C05383=1024.607,74.316,-103.652,167.758,48.129,158.923
C05384=1024.602,74.066,-103.634,167.757,48.134,158.924
C05385=1024.596,73.817,-103.616,167.754,48.137,158.924
C05386=1024.590,73.567,-103.600,167.751,48.141,158.924
C05387=1024.584,73.318,-103.582,167.749,48.146,158.925
C05388=1024.578,73.069,-103.565,167.746,48.150,158.925
C05389=1024.572,72.819,-103.547,167.743,48.154,158.926
C05390=1024.566,72.570,-103.530,167.740,48.157,158.926
C05391=1024.560,72.321,-103.512,167.739,48.162,158.926
C05392=1024.554,72.071,-103.494,167.736,48.166,158.927
C05393=1024.548,71.823,-103.477,167.733,48.169,158.927
C05394=1024.542,71.572,-103.460,167.730,48.173,158.928
C05395=1024.537,71.323,-103.443,167.728,48.178,158.928
C05396=1024.531,71.074,-103.425,167.725,48.182,158.928
C05397=1024.524,70.825,-103.408,167.723,48.185,158.929
C05398=1024.519,70.576,-103.390,167.721,48.190,158.929
C05399=1024.513,70.327,-103.372,167.718,48.194,158.930
C05400=1024.507,70.077,-103.356,167.715,48.197,158.930
C05401=1024.501,69.828,-103.338,167.712,48.201,158.930
C05402=1024.495,69.578,-103.320,167.710,48.206,158.931
C05403=1024.489,69.329,-103.303,167.708,48.209,158.931
C05404=1024.483,69.080,-103.286,167.705,48.213,158.932
C05405=1024.477,68.830,-103.269,167.702,48.217,158.932
C05406=1024.472,68.581,-103.251,167.700,48.222,158.933
C05407=1024.466,68.332,-103.234,167.697,48.226,158.933
C05408=1024.460,68.082,-103.217,167.694,48.229,158.933
C05409=1024.454,67.833,-103.200,167.692,48.234,158.934
C05410=1024.448,67.584,-103.182,167.690,48.238,158.934
C05411=1024.441,67.334,-103.165,167.687,48.241,158.935
C05412=1024.436,67.085,-103.148,167.684,48.245,158.935
C05413=1024.430,66.836,-103.131,167.682,48.250,158.935
C05414=1024.424,66.586,-103.113,167.679,48.254,158.936
C05415=1024.418,66.337,-103.097,167.676,48.258,158.936
C05416=1024.412,66.088,-103.079,167.674,48.262,158.937
C05417=1024.406,65.837,-103.062,167.672,48.266,158.937
C05418=1024.400,65.589,-103.045,167.669,48.270,158.937
C05419=1024.394,65.340,-103.028,167.667,48.274,158.938
C05420=1024.388,65.090,-103.011,167.664,48.278,158.938
C05421=1024.382,64.841,-102.993,167.661,48.282,158.939
C05422=1024.376,64.592,-102.976,167.658,48.286,158.939
C05423=1024.370,64.342,-102.959,167.656,48.290,158.940
C05424=1024.364,64.093,-102.942,167.654,48.294,158.940
C05425=1024.359,63.843,-102.925,167.651,48.298,158.940
C05426=1024.352,63.594,-102.908,167.649,48.302,158.941
C05427=1024.347,63.344,-102.891,167.646,48.306,158.941
C05428=1024.341,63.095,-102.874,167.643,48.310,158.942
C05429=1024.334,62.845,-102.858,167.641,48.315,158.942
C05430=1024.328,62.597,-102.841,167.638,48.319,158.942
C05431=1024.323,62.347,-102.824,167.635,48.323,158.943
C05432=1024.317,62.098,-102.808,167.633,48.327,158.943
C05433=1024.310,61.848,-102.790,167.631,48.331,158.944
C05434=1024.304,61.599,-102.774,167.628,48.335,158.944
C05435=1024.298,61.350,-102.757,167.626,48.339,158.945
C05436=1024.292,61.100,-102.740,167.623,48.344,158.945
C05437=1024.285,60.851,-102.723,167.620,48.347,158.945
C05438=1024.279,60.602,-102.707,167.618,48.352,158.946
C05439=1024.274,60.352,-102.690,167.615,48.356,158.946
C05440=1024.267,60.103,-102.673,167.612,48.360,158.947
C05441=1024.260,59.819,-102.654,167.610,48.364,158.947
C05442=1024.253,59.534,-102.635,167.606,48.369,158.948
C05443=1024.246,59.249,-102.616,167.604,48.374,158.948
C05444=1024.240,58.965,-102.596,167.600,48.379,158.948
C05445=1024.234,58.716,-102.580,167.598,48.383,158.949
C05446=1024.227,58.466,-102.564,167.595,48.387,158.949
C05447=1024.221,58.217,-102.547,167.594,48.391,158.950
C05448=1024.215,57.967,-102.530,167.591,48.395,158.950
C05449=1024.209,57.718,-102.514,167.588,48.399,158.951
C05450=1024.204,57.469,-102.497,167.585,48.404,158.951
C05451=1024.197,57.219,-102.480,167.583,48.408,158.952
C05452=1024.191,56.970,-102.464,167.580,48.412,158.952
C05453=1024.185,56.721,-102.447,167.577,48.416,158.952
C05454=1024.179,56.472,-102.430,167.575,48.420,158.953
C05455=1024.174,56.222,-102.414,167.572,48.424,158.953
C05456=1024.167,55.972,-102.397,167.569,48.428,158.954
C05457=1024.161,55.723,-102.380,167.568,48.432,158.954
C05458=1024.155,55.474,-102.364,167.565,48.436,158.954
C05459=1024.149,55.224,-102.347,167.562,48.441,158.955
C05460=1024.143,54.975,-102.331,167.560,48.444,158.955
C05461=1024.137,54.725,-102.313,167.557,48.448,158.956
C05462=1024.131,54.476,-102.297,167.554,48.453,158.956
C05463=1024.125,54.227,-102.281,167.551,48.457,158.956
C05464=1024.119,53.977,-102.264,167.549,48.461,158.957
C05465=1024.113,53.728,-102.248,167.547,48.465,158.957
C05466=1024.107,53.479,-102.231,167.544,48.469,158.958
C05467=1024.102,53.230,-102.214,167.542,48.473,158.958
C05468=1024.095,52.980,-102.198,167.539,48.477,158.958
C05469=1024.089,52.730,-102.182,167.536,48.481,158.959
C05470=1024.083,52.481,-102.165,167.534,48.485,158.959
C05471=1024.077,52.232,-102.148,167.531,48.489,158.960
C05472=1024.071,51.983,-102.132,167.528,48.494,158.960
C05473=1024.066,51.733,-102.115,167.527,48.497,158.961
C05474=1024.060,51.484,-102.099,167.524,48.501,158.961
C05475=1024.054,51.234,-102.083,167.521,48.505,158.961
C05476=1024.048,50.985,-102.066,167.519,48.510,158.962
C05477=1024.041,50.735,-102.050,167.516,48.513,158.962
C05478=1024.035,50.486,-102.033,167.513,48.517,158.962
C05479=1024.030,50.237,-102.016,167.510,48.521,158.963
C05480=1024.024,49.987,-102.000,167.508,48.525,158.963
C05481=1024.018,49.738,-101.983,167.506,48.529,158.964
C05482=1024.012,49.489,-101.967,167.503,48.533,158.964
C05483=1024.006,49.239,-101.951,167.500,48.537,158.964
C05484=1024.000,48.990,-101.935,167.498,48.541,158.965
C05485=1023.995,48.740,-101.918,167.495,48.546,158.965
C05486=1023.989,48.491,-101.902,167.493,48.549,158.966
C05487=1023.983,48.242,-101.885,167.491,48.553,158.966
C05488=1023.977,47.992,-101.869,167.488,48.557,158.966
C05489=1023.971,47.743,-101.853,167.485,48.561,158.967
C05490=1023.965,47.494,-101.836,167.483,48.566,158.967
C05491=1023.959,47.245,-101.820,167.480,48.570,158.968
C05492=1023.954,46.995,-101.803,167.478,48.573,158.968
C05493=1023.948,46.746,-101.786,167.475,48.577,158.968
C05494=1023.942,46.496,-101.770,167.472,48.581,158.969
C05495=1023.935,46.246,-101.754,167.470,48.585,158.969
C05496=1023.929,45.997,-101.737,167.467,48.589,158.969
C05497=1023.923,45.748,-101.721,167.464,48.593,158.970
C05498=1023.917,45.498,-101.705,167.463,48.597,158.970
C05499=1023.912,45.249,-101.688,167.460,48.601,158.971
C05500=1023.906,44.999,-101.672,167.457,48.605,158.971
C05501=1023.901,44.751,-101.656,167.454,48.609,158.971
C05502=1023.895,44.501,-101.640,167.452,48.613,158.972
C05503=1023.889,44.252,-101.623,167.449,48.617,158.972
C05504=1023.883,44.003,-101.607,167.447,48.621,158.973
C05505=1023.876,43.717,-101.589,167.444,48.625,158.973
C05506=1023.870,43.433,-101.570,167.441,48.630,158.973
C05507=1023.863,43.148,-101.551,167.439,48.634,158.974
C05508=1023.857,42.863,-101.533,167.435,48.638,158.974
C05509=1023.851,42.614,-101.516,167.432,48.642,158.974
C05510=1023.845,42.364,-101.501,167.431,48.647,158.975
C05511=1023.839,42.115,-101.484,167.428,48.651,158.975
C05512=1023.833,41.865,-101.469,167.425,48.654,158.976
C05513=1023.827,41.616,-101.453,167.422,48.658,158.976
C05514=1023.821,41.366,-101.436,167.420,48.663,158.977
C05515=1023.815,41.117,-101.420,167.417,48.667,158.977
C05516=1023.809,40.868,-101.404,167.414,48.671,158.977
C05517=1023.804,40.618,-101.388,167.412,48.675,158.978
C05518=1023.797,40.369,-101.373,167.409,48.679,158.978
C05519=1023.791,40.119,-101.356,167.407,48.683,158.978
C05520=1023.785,39.870,-101.340,167.405,48.687,158.979
C05521=1023.779,39.620,-101.325,167.402,48.691,158.979
C05522=1023.773,39.371,-101.308,167.399,48.695,158.980
C05523=1023.767,39.121,-101.292,167.397,48.699,158.980
C05524=1023.761,38.872,-101.276,167.394,48.703,158.980
C05525=1023.756,38.623,-101.261,167.391,48.707,158.981
C05526=1023.750,38.374,-101.245,167.388,48.711,158.981
C05527=1023.744,38.124,-101.229,167.387,48.715,158.982
C05528=1023.738,37.874,-101.213,167.384,48.719,158.982
C05529=1023.732,37.625,-101.197,167.381,48.723,158.982
C05530=1023.726,37.376,-101.181,167.378,48.727,158.983
C05531=1023.720,37.126,-101.166,167.376,48.731,158.983
C05532=1023.714,36.877,-101.150,167.373,48.736,158.983
C05533=1023.708,36.627,-101.133,167.370,48.740,158.984
C05534=1023.702,36.377,-101.118,167.368,48.744,158.984
C05535=1023.696,36.129,-101.102,167.365,48.747,158.984
C05536=1023.691,35.879,-101.087,167.363,48.752,158.985
C05537=1023.684,35.630,-101.071,167.361,48.756,158.985
C05538=1023.678,35.380,-101.056,167.358,48.760,158.986
C05539=1023.672,35.131,-101.039,167.356,48.764,158.986
C05540=1023.666,34.881,-101.025,167.353,48.768,158.987
C05541=1023.660,34.632,-101.008,167.350,48.772,158.987
C05542=1023.654,34.382,-100.993,167.348,48.777,158.987
C05543=1023.648,34.133,-100.977,167.345,48.781,158.988
C05544=1023.643,33.883,-100.962,167.342,48.785,158.988
C05545=1023.636,33.634,-100.946,167.339,48.789,158.988
C05546=1023.630,33.384,-100.931,167.337,48.793,158.989
C05547=1023.624,33.135,-100.915,167.334,48.797,158.989
C05548=1023.618,32.885,-100.899,167.331,48.801,158.990
C05549=1023.612,32.636,-100.883,167.329,48.805,158.990
C05550=1023.606,32.387,-100.869,167.327,48.809,158.991
C05551=1023.600,32.138,-100.852,167.324,48.813,158.991
C05552=1023.594,31.888,-100.837,167.322,48.817,158.991
C05553=1023.588,31.639,-100.821,167.319,48.821,158.992
C05554=1023.582,31.389,-100.806,167.316,48.826,158.992
C05555=1023.576,31.141,-100.790,167.314,48.830,158.992
C05556=1023.571,30.891,-100.775,167.311,48.834,158.993
C05557=1023.564,30.641,-100.760,167.308,48.837,158.993
C05558=1023.558,30.392,-100.744,167.305,48.841,158.993
C05559=1023.553,30.142,-100.728,167.303,48.846,158.994
C05560=1023.546,29.893,-100.713,167.300,48.850,158.994
C05561=1023.541,29.643,-100.697,167.298,48.854,158.995
C05562=1023.534,29.394,-100.682,167.296,48.858,158.995
C05563=1023.528,29.144,-100.666,167.293,48.861,158.995
C05564=1023.523,28.894,-100.650,167.290,48.866,158.996
C05565=1023.517,28.645,-100.636,167.288,48.870,158.996
C05566=1023.511,28.396,-100.620,167.285,48.874,158.996
C05567=1023.505,28.146,-100.605,167.282,48.878,158.997
C05568=1023.499,27.897,-100.588,167.279,48.882,158.997
C05569=1023.492,27.612,-100.572,167.277,48.887,158.998
C05570=1023.485,27.327,-100.555,167.273,48.891,158.998
C05571=1023.479,27.043,-100.537,167.271,48.896,158.999
C05572=1023.472,26.758,-100.519,167.268,48.901,158.999
C05573=1023.466,26.508,-100.504,167.265,48.905,158.999
C05574=1023.460,26.259,-100.488,167.262,48.909,159.000
C05575=1023.453,26.009,-100.473,167.259,48.913,159.000
C05576=1023.448,25.760,-100.458,167.257,48.917,159.000
C05577=1023.442,25.510,-100.443,167.255,48.921,159.001
C05578=1023.435,25.261,-100.427,167.252,48.925,159.001
C05579=1023.430,25.011,-100.412,167.250,48.929,159.002
C05580=1023.424,24.762,-100.397,167.247,48.934,159.002
C05581=1023.417,24.513,-100.382,167.244,48.938,159.002
C05582=1023.412,24.263,-100.367,167.242,48.942,159.003
C05583=1023.406,24.014,-100.352,167.239,48.945,159.003
C05584=1023.399,23.765,-100.337,167.237,48.950,159.004
C05585=1023.394,23.515,-100.321,167.234,48.954,159.004
C05586=1023.388,23.266,-100.306,167.231,48.958,159.004
C05587=1023.381,23.016,-100.291,167.228,48.962,159.005
C05588=1023.376,22.766,-100.276,167.226,48.967,159.005
C05589=1023.369,22.517,-100.261,167.223,48.971,159.005
C05590=1023.364,22.268,-100.246,167.220,48.974,159.006
C05591=1023.358,22.018,-100.231,167.218,48.978,159.006
C05592=1023.352,21.768,-100.216,167.215,48.982,159.006
C05593=1023.346,21.520,-100.201,167.212,48.987,159.007
C05594=1023.340,21.270,-100.185,167.210,48.991,159.007
C05595=1023.334,21.020,-100.170,167.207,48.995,159.008
C05596=1023.328,20.771,-100.156,167.205,48.999,159.008
C05597=1023.322,20.521,-100.140,167.202,49.003,159.008
C05598=1023.316,20.272,-100.125,167.200,49.006,159.009
C05599=1023.310,20.023,-100.110,167.197,49.011,159.009
C05600=1023.304,19.773,-100.095,167.194,49.015,159.009
C05601=1023.299,19.524,-100.080,167.192,49.019,159.010
C05602=1023.292,19.274,-100.065,167.189,49.023,159.010
C05603=1023.286,19.024,-100.050,167.186,49.027,159.010
C05604=1023.281,18.775,-100.035,167.184,49.032,159.011
C05605=1023.274,18.525,-100.020,167.181,49.036,159.011
C05606=1023.268,18.276,-100.005,167.178,49.039,159.012
C05607=1023.262,18.027,-99.991,167.175,49.043,159.012
C05608=1023.257,17.777,-99.975,167.173,49.047,159.012
C05609=1023.251,17.528,-99.961,167.170,49.052,159.013
C05610=1023.245,17.278,-99.946,167.168,49.056,159.013
C05611=1023.238,17.028,-99.932,167.165,49.060,159.013
C05612=1023.232,16.779,-99.917,167.162,49.064,159.014
C05613=1023.226,16.529,-99.902,167.160,49.069,159.014
C05614=1023.221,16.280,-99.887,167.157,49.073,159.015
C05615=1023.215,16.030,-99.872,167.154,49.077,159.015
C05616=1023.209,15.781,-99.857,167.151,49.080,159.015
C05617=1023.203,15.532,-99.842,167.149,49.084,159.015
C05618=1023.196,15.282,-99.827,167.146,49.088,159.016
C05619=1023.191,15.032,-99.813,167.144,49.093,159.016
C05620=1023.185,14.783,-99.798,167.142,49.097,159.017
C05621=1023.179,14.534,-99.783,167.139,49.101,159.017
C05622=1023.173,14.284,-99.768,167.136,49.105,159.017
C05623=1023.167,14.035,-99.754,167.134,49.109,159.018
C05624=1023.161,13.785,-99.739,167.131,49.113,159.018
C05625=1023.156,13.535,-99.724,167.128,49.117,159.018
C05626=1023.150,13.286,-99.710,167.126,49.121,159.019
C05627=1023.142,13.036,-99.695,167.123,49.125,159.019
C05628=1023.137,12.787,-99.681,167.120,49.129,159.020
C05629=1023.131,12.537,-99.666,167.118,49.134,159.020
C05630=1023.125,12.288,-99.652,167.115,49.138,159.020
C05631=1023.119,12.038,-99.638,167.112,49.142,159.021
C05632=1023.113,11.789,-99.623,167.109,49.147,159.021
C05633=1023.106,11.506,-99.607,167.106,49.151,159.021
C05634=1023.099,11.222,-99.590,167.103,49.156,159.022
C05635=1023.092,10.939,-99.574,167.100,49.160,159.022
C05636=1023.085,10.656,-99.558,167.097,49.165,159.023
C05637=1023.079,10.406,-99.543,167.094,49.169,159.023
C05638=1023.073,10.157,-99.528,167.092,49.174,159.024
C05639=1023.067,9.907,-99.514,167.089,49.178,159.024
C05640=1023.061,9.658,-99.500,167.086,49.182,159.024
C05641=1023.055,9.408,-99.485,167.083,49.186,159.024
C05642=1023.049,9.159,-99.471,167.081,49.190,159.025
C05643=1023.043,8.909,-99.456,167.078,49.194,159.025
C05644=1023.037,8.660,-99.442,167.076,49.198,159.026
C05645=1023.030,8.410,-99.428,167.073,49.202,159.026
C05646=1023.025,8.161,-99.414,167.070,49.207,159.026
C05647=1023.018,7.911,-99.399,167.068,49.211,159.027
C05648=1023.013,7.662,-99.384,167.065,49.215,159.027
C05649=1023.007,7.412,-99.370,167.062,49.219,159.027
C05650=1023.001,7.163,-99.355,167.059,49.223,159.028
C05651=1022.995,6.913,-99.341,167.057,49.228,159.028
C05652=1022.989,6.664,-99.327,167.054,49.232,159.029
C05653=1022.984,6.414,-99.313,167.052,49.236,159.029
C05654=1022.976,6.165,-99.298,167.049,49.240,159.029
C05655=1022.971,5.915,-99.285,167.046,49.244,159.030
C05656=1022.965,5.665,-99.270,167.044,49.248,159.030
C05657=1022.959,5.416,-99.256,167.041,49.252,159.030
C05658=1022.953,5.167,-99.241,167.038,49.256,159.031
C05659=1022.947,4.917,-99.227,167.035,49.260,159.031
C05660=1022.941,4.668,-99.212,167.033,49.264,159.031
C05661=1022.935,4.417,-99.198,167.030,49.268,159.032
C05662=1022.929,4.169,-99.184,167.027,49.272,159.032
C05663=1022.923,3.919,-99.170,167.025,49.277,159.032
C05664=1022.917,3.669,-99.156,167.022,49.281,159.033
C05665=1022.911,3.420,-99.141,167.019,49.285,159.033
C05666=1022.905,3.170,-99.127,167.017,49.289,159.033
C05667=1022.900,2.921,-99.113,167.014,49.293,159.034
C05668=1022.894,2.671,-99.099,167.011,49.297,159.034
C05669=1022.887,2.421,-99.085,167.008,49.301,159.034
C05670=1022.882,2.172,-99.071,167.006,49.305,159.035
C05671=1022.876,1.923,-99.057,167.003,49.309,159.035
C05672=1022.870,1.673,-99.042,167.001,49.313,159.035
C05673=1022.864,1.423,-99.028,166.998,49.317,159.036
C05674=1022.859,1.174,-99.014,166.995,49.321,159.036
C05675=1022.852,0.924,-98.999,166.992,49.325,159.036
C05676=1022.846,0.675,-98.986,166.990,49.329,159.037
C05677=1022.841,0.425,-98.972,166.987,49.333,159.037
C05678=1022.834,0.176,-98.957,166.984,49.337,159.037
C05679=1022.829,-0.074,-98.943,166.981,49.341,159.038
C05680=1022.823,-0.324,-98.929,166.979,49.345,159.038
C05681=1022.818,-0.572,-98.915,166.976,49.349,159.038
C05682=1022.811,-0.823,-98.900,166.973,49.353,159.039
C05683=1022.805,-1.072,-98.887,166.970,49.357,159.039
C05684=1022.799,-1.321,-98.873,166.968,49.361,159.039
C05685=1022.793,-1.571,-98.858,166.965,49.365,159.040
C05686=1022.788,-1.821,-98.845,166.962,49.369,159.040
C05687=1022.782,-2.070,-98.830,166.960,49.373,159.040
C05688=1022.777,-2.319,-98.816,166.957,49.377,159.041
C05689=1022.771,-2.570,-98.802,166.954,49.381,159.041
C05690=1022.764,-2.819,-98.789,166.951,49.385,159.041
C05691=1022.759,-3.068,-98.774,166.949,49.389,159.042
C05692=1022.753,-3.317,-98.760,166.946,49.393,159.042
C05693=1022.747,-3.568,-98.746,166.943,49.397,159.042
C05694=1022.742,-3.817,-98.732,166.940,49.401,159.042
C05695=1022.736,-4.067,-98.718,166.938,49.405,159.043
C05696=1022.730,-4.315,-98.704,166.935,49.410,159.043
C05697=1022.722,-4.598,-98.689,166.932,49.414,159.043
C05698=1022.715,-4.879,-98.673,166.928,49.419,159.044
C05699=1022.709,-5.161,-98.658,166.926,49.424,159.044
C05700=1022.702,-5.442,-98.642,166.922,49.429,159.045
C05701=1022.696,-5.691,-98.628,166.920,49.433,159.045
C05702=1022.690,-5.941,-98.615,166.917,49.437,159.045
C05703=1022.685,-6.190,-98.601,166.914,49.441,159.046
C05704=1022.678,-6.440,-98.588,166.911,49.445,159.046
C05705=1022.672,-6.690,-98.574,166.909,49.449,159.047
C05706=1022.666,-6.939,-98.561,166.906,49.453,159.047
C05707=1022.661,-7.189,-98.547,166.904,49.457,159.047
C05708=1022.655,-7.438,-98.533,166.900,49.462,159.047
C05709=1022.648,-7.688,-98.519,166.897,49.466,159.048
C05710=1022.642,-7.937,-98.506,166.894,49.470,159.048
C05711=1022.637,-8.187,-98.492,166.892,49.474,159.048
C05712=1022.631,-8.436,-98.479,166.889,49.478,159.049
C05713=1022.625,-8.686,-98.465,166.887,49.482,159.049
C05714=1022.619,-8.935,-98.452,166.884,49.486,159.049
C05715=1022.613,-9.185,-98.437,166.881,49.490,159.050
C05716=1022.607,-9.435,-98.424,166.878,49.495,159.050
C05717=1022.601,-9.685,-98.411,166.876,49.499,159.050
C05718=1022.595,-9.934,-98.398,166.873,49.503,159.051
C05719=1022.590,-10.184,-98.384,166.871,49.507,159.051
C05720=1022.583,-10.433,-98.371,166.867,49.512,159.051
C05721=1022.577,-10.682,-98.357,166.864,49.516,159.052
C05722=1022.571,-10.933,-98.343,166.861,49.520,159.052
C05723=1022.565,-11.182,-98.330,166.859,49.524,159.052
C05724=1022.559,-11.431,-98.316,166.856,49.528,159.053
C05725=1022.553,-11.681,-98.303,166.853,49.532,159.053
C05726=1022.548,-11.930,-98.289,166.851,49.536,159.053
C05727=1022.542,-12.180,-98.276,166.848,49.540,159.054
C05728=1022.536,-12.430,-98.262,166.845,49.544,159.054
C05729=1022.530,-12.679,-98.249,166.842,49.548,159.054
C05730=1022.525,-12.928,-98.235,166.840,49.552,159.054
C05731=1022.518,-13.178,-98.222,166.837,49.556,159.055
C05732=1022.512,-13.428,-98.208,166.835,49.560,159.055
C05733=1022.507,-13.678,-98.195,166.832,49.564,159.056
C05734=1022.501,-13.928,-98.181,166.828,49.569,159.056
C05735=1022.495,-14.177,-98.168,166.825,49.573,159.056
C05736=1022.489,-14.426,-98.155,166.823,49.577,159.056
C05737=1022.483,-14.676,-98.141,166.820,49.581,159.057
C05738=1022.477,-14.925,-98.128,166.817,49.585,159.057
C05739=1022.472,-15.175,-98.115,166.814,49.589,159.057
C05740=1022.466,-15.424,-98.101,166.812,49.593,159.058
C05741=1022.460,-15.674,-98.087,166.809,49.597,159.058
C05742=1022.454,-15.924,-98.075,166.806,49.601,159.058
C05743=1022.448,-16.173,-98.062,166.804,49.605,159.059
C05744=1022.442,-16.422,-98.048,166.801,49.609,159.059
C05745=1022.437,-16.673,-98.035,166.797,49.613,159.059
C05746=1022.430,-16.922,-98.022,166.795,49.618,159.060
C05747=1022.424,-17.172,-98.009,166.792,49.622,159.060
C05748=1022.418,-17.421,-97.996,166.789,49.626,159.060
C05749=1022.412,-17.670,-97.983,166.787,49.630,159.061
C05750=1022.407,-17.920,-97.970,166.784,49.634,159.061
C05751=1022.401,-18.170,-97.956,166.781,49.638,159.061
C05752=1022.395,-18.420,-97.944,166.777,49.642,159.061
C05753=1022.389,-18.669,-97.931,166.775,49.647,159.062
C05754=1022.383,-18.919,-97.918,166.772,49.651,159.062
C05755=1022.377,-19.168,-97.904,166.770,49.655,159.062
C05756=1022.371,-19.417,-97.891,166.767,49.659,159.063
C05757=1022.365,-19.667,-97.878,166.764,49.663,159.063
C05758=1022.359,-19.917,-97.865,166.762,49.667,159.063
C05759=1022.353,-20.167,-97.852,166.758,49.671,159.064
C05760=1022.347,-20.416,-97.839,166.755,49.675,159.064
C05761=1022.340,-20.696,-97.824,166.753,49.680,159.064
C05762=1022.334,-20.976,-97.809,166.749,49.685,159.065
C05763=1022.327,-21.255,-97.795,166.746,49.690,159.065
C05764=1022.320,-21.535,-97.780,166.743,49.694,159.065
C05765=1022.314,-21.785,-97.768,166.740,49.698,159.066
C05766=1022.309,-22.035,-97.755,166.738,49.702,159.066
C05767=1022.302,-22.284,-97.742,166.734,49.707,159.066
C05768=1022.297,-22.533,-97.730,166.731,49.711,159.067
C05769=1022.292,-22.783,-97.716,166.729,49.715,159.067
C05770=1022.286,-23.033,-97.703,166.726,49.719,159.067
C05771=1022.279,-23.282,-97.690,166.723,49.723,159.067
C05772=1022.274,-23.532,-97.677,166.720,49.727,159.068
C05773=1022.267,-23.781,-97.664,166.718,49.731,159.068
C05774=1022.261,-24.031,-97.652,166.715,49.735,159.068
C05775=1022.256,-24.281,-97.638,166.711,49.739,159.069
C05776=1022.250,-24.530,-97.625,166.709,49.743,159.069
C05777=1022.244,-24.780,-97.613,166.706,49.747,159.069
C05778=1022.238,-25.029,-97.600,166.703,49.751,159.069
C05779=1022.233,-25.279,-97.587,166.700,49.755,159.070
C05780=1022.227,-25.529,-97.575,166.698,49.759,159.070
C05781=1022.221,-25.778,-97.561,166.695,49.763,159.070
C05782=1022.215,-26.028,-97.548,166.692,49.767,159.071
C05783=1022.209,-26.278,-97.536,166.689,49.772,159.071
C05784=1022.204,-26.527,-97.523,166.686,49.776,159.071
C05785=1022.198,-26.776,-97.510,166.683,49.780,159.072
C05786=1022.192,-27.026,-97.498,166.681,49.784,159.072
C05787=1022.186,-27.276,-97.484,166.678,49.788,159.072
C05788=1022.181,-27.526,-97.471,166.675,49.792,159.072
C05789=1022.175,-27.776,-97.459,166.672,49.796,159.073
C05790=1022.168,-28.025,-97.447,166.669,49.800,159.073
C05791=1022.163,-28.274,-97.435,166.666,49.804,159.073
C05792=1022.156,-28.524,-97.421,166.664,49.809,159.074
C05793=1022.151,-28.774,-97.409,166.661,49.813,159.074
C05794=1022.145,-29.023,-97.396,166.658,49.817,159.074
C05795=1022.139,-29.273,-97.384,166.654,49.822,159.074
C05796=1022.133,-29.523,-97.371,166.652,49.826,159.075
C05797=1022.128,-29.772,-97.359,166.649,49.830,159.075
C05798=1022.122,-30.022,-97.346,166.646,49.834,159.075
C05799=1022.115,-30.271,-97.334,166.644,49.838,159.076
C05800=1022.109,-30.521,-97.321,166.641,49.842,159.076
C05801=1022.103,-30.770,-97.309,166.638,49.847,159.076
C05802=1022.098,-31.020,-97.296,166.635,49.851,159.077
C05803=1022.092,-31.270,-97.284,166.632,49.855,159.077
C05804=1022.086,-31.520,-97.271,166.629,49.859,159.077
C05805=1022.080,-31.770,-97.259,166.627,49.863,159.078
C05806=1022.075,-32.019,-97.246,166.623,49.867,159.078
C05807=1022.068,-32.269,-97.235,166.620,49.871,159.078
C05808=1022.062,-32.518,-97.222,166.618,49.875,159.078
C05809=1022.057,-32.768,-97.210,166.615,49.880,159.079
C05810=1022.051,-33.018,-97.197,166.612,49.884,159.079
C05811=1022.045,-33.267,-97.184,166.608,49.888,159.079
C05812=1022.039,-33.517,-97.171,166.606,49.892,159.079
C05813=1022.033,-33.766,-97.159,166.603,49.896,159.080
C05814=1022.027,-34.015,-97.147,166.600,49.900,159.080
C05815=1022.021,-34.265,-97.135,166.598,49.904,159.080
C05816=1022.015,-34.514,-97.123,166.594,49.908,159.081
C05817=1022.010,-34.764,-97.110,166.591,49.913,159.081
C05818=1022.004,-35.014,-97.097,166.589,49.917,159.081
C05819=1021.998,-35.263,-97.085,166.586,49.921,159.081
C05820=1021.992,-35.513,-97.073,166.583,49.925,159.082
C05821=1021.986,-35.764,-97.061,166.580,49.929,159.082
C05822=1021.981,-36.013,-97.049,166.577,49.933,159.082
C05823=1021.975,-36.263,-97.037,166.574,49.937,159.083
C05824=1021.969,-36.512,-97.024,166.571,49.941,159.083
C05825=1021.962,-36.791,-97.011,166.568,49.946,159.083
C05826=1021.956,-37.070,-96.996,166.565,49.950,159.084
C05827=1021.949,-37.349,-96.983,166.562,49.955,159.084
C05828=1021.943,-37.627,-96.969,166.558,49.960,159.084
C05829=1021.938,-37.878,-96.957,166.555,49.964,159.084
C05830=1021.932,-38.127,-96.945,166.553,49.968,159.085
C05831=1021.926,-38.376,-96.933,166.550,49.972,159.085
C05832=1021.920,-38.626,-96.920,166.547,49.976,159.085
C05833=1021.915,-38.876,-96.908,166.545,49.980,159.086
C05834=1021.909,-39.125,-96.895,166.541,49.984,159.086
C05835=1021.903,-39.375,-96.883,166.538,49.988,159.086
C05836=1021.897,-39.625,-96.872,166.536,49.993,159.086
C05837=1021.891,-39.875,-96.859,166.533,49.997,159.087
C05838=1021.885,-40.124,-96.848,166.529,50.001,159.087
C05839=1021.880,-40.374,-96.836,166.526,50.005,159.087
C05840=1021.873,-40.624,-96.824,166.524,50.009,159.087
C05841=1021.868,-40.873,-96.812,166.521,50.013,159.088
C05842=1021.862,-41.123,-96.799,166.517,50.018,159.088
C05843=1021.856,-41.372,-96.788,166.515,50.022,159.088
C05844=1021.850,-41.622,-96.776,166.512,50.026,159.089
C05845=1021.844,-41.871,-96.764,166.510,50.030,159.089
C05846=1021.838,-42.121,-96.753,166.506,50.035,159.089
C05847=1021.832,-42.371,-96.740,166.503,50.039,159.089
C05848=1021.826,-42.620,-96.728,166.501,50.043,159.090
C05849=1021.821,-42.871,-96.717,166.498,50.047,159.090
C05850=1021.815,-43.120,-96.705,166.494,50.051,159.090
C05851=1021.809,-43.369,-96.692,166.491,50.055,159.091
C05852=1021.803,-43.619,-96.681,166.489,50.059,159.091
C05853=1021.797,-43.869,-96.669,166.486,50.064,159.091
C05854=1021.792,-44.119,-96.657,166.483,50.068,159.091
C05855=1021.786,-44.368,-96.646,166.480,50.072,159.092
C05856=1021.780,-44.617,-96.633,166.477,50.076,159.092
C05857=1021.774,-44.868,-96.622,166.474,50.080,159.092
C05858=1021.769,-45.117,-96.610,166.472,50.084,159.092
C05859=1021.762,-45.367,-96.599,166.468,50.089,159.093
C05860=1021.757,-45.616,-96.586,166.465,50.093,159.093
C05861=1021.751,-45.866,-96.575,166.462,50.097,159.093
C05862=1021.745,-46.115,-96.563,166.460,50.101,159.094
C05863=1021.740,-46.366,-96.551,166.456,50.105,159.094
C05864=1021.734,-46.615,-96.540,166.453,50.109,159.094
C05865=1021.728,-46.865,-96.527,166.451,50.113,159.094
C05866=1021.722,-47.114,-96.516,166.448,50.117,159.095
C05867=1021.717,-47.363,-96.504,166.445,50.121,159.095
C05868=1021.710,-47.614,-96.493,166.442,50.126,159.095
C05869=1021.705,-47.863,-96.481,166.439,50.130,159.095
C05870=1021.699,-48.113,-96.469,166.436,50.134,159.096
C05871=1021.693,-48.362,-96.457,166.434,50.138,159.096
C05872=1021.688,-48.613,-96.445,166.430,50.142,159.096
C05873=1021.682,-48.862,-96.434,166.427,50.147,159.096
C05874=1021.677,-49.111,-96.422,166.424,50.150,159.097
C05875=1021.670,-49.362,-96.411,166.421,50.154,159.097
C05876=1021.665,-49.611,-96.399,166.419,50.158,159.097
C05877=1021.659,-49.861,-96.388,166.415,50.162,159.097
C05878=1021.653,-50.110,-96.375,166.412,50.167,159.098
C05879=1021.648,-50.360,-96.364,166.410,50.171,159.098
C05880=1021.642,-50.610,-96.353,166.407,50.175,159.098
C05881=1021.636,-50.859,-96.341,166.403,50.179,159.098
C05882=1021.631,-51.109,-96.330,166.401,50.183,159.099
C05883=1021.625,-51.359,-96.318,166.398,50.187,159.099
C05884=1021.619,-51.608,-96.307,166.394,50.192,159.099
C05885=1021.612,-51.858,-96.295,166.392,50.196,159.099
C05886=1021.607,-52.107,-96.285,166.389,50.201,159.100
C05887=1021.602,-52.357,-96.273,166.385,50.205,159.100
C05888=1021.595,-52.607,-96.262,166.383,50.209,159.100
C05889=1021.589,-52.855,-96.251,166.380,50.213,159.101
C05890=1021.583,-53.103,-96.239,166.376,50.217,159.101
C05891=1021.578,-53.350,-96.229,166.374,50.222,159.101
C05892=1021.572,-53.597,-96.217,166.371,50.226,159.101
C05893=1021.566,-53.845,-96.206,166.368,50.231,159.102
C05894=1021.560,-54.093,-96.195,166.365,50.235,159.102
C05895=1021.554,-54.341,-96.185,166.362,50.239,159.102
C05896=1021.548,-54.589,-96.173,166.360,50.243,159.103
C05897=1021.543,-54.838,-96.162,166.356,50.247,159.103
C05898=1021.537,-55.088,-96.151,166.353,50.251,159.103
C05899=1021.531,-55.338,-96.140,166.351,50.256,159.103
C05900=1021.525,-55.587,-96.129,166.347,50.260,159.103
C05901=1021.520,-55.837,-96.117,166.344,50.264,159.104
C05902=1021.514,-56.087,-96.106,166.342,50.268,159.104
C05903=1021.508,-56.337,-96.095,166.338,50.273,159.104
C05904=1021.502,-56.586,-96.084,166.335,50.277,159.105
C05905=1021.496,-56.835,-96.073,166.333,50.281,159.105
C05906=1021.490,-57.085,-96.062,166.329,50.286,159.105
C05907=1021.484,-57.335,-96.051,166.326,50.290,159.105
C05908=1021.478,-57.584,-96.040,166.324,50.294,159.106
C05909=1021.472,-57.868,-96.027,166.320,50.299,159.106
C05910=1021.465,-58.151,-96.015,166.317,50.304,159.106
C05911=1021.459,-58.434,-96.002,166.313,50.309,159.107
C05912=1021.452,-58.717,-95.990,166.310,50.313,159.107
C05913=1021.447,-58.968,-95.978,166.307,50.317,159.107
C05914=1021.441,-59.217,-95.967,166.303,50.322,159.107
///RCONF 1,0,0,1,0,0,0,0,0,0,0,0,0,0,0,0,0,0,0,0,0,0,0,0
C05915=1021.435,-59.467,-95.956,166.301,50.326,159.108
C05916=1021.429,-59.716,-95.945,166.298,50.330,159.108
C05917=1021.424,-59.966,-95.935,166.294,50.334,159.108
C05918=1021.417,-60.216,-95.923,166.292,50.338,159.108
C05919=1021.411,-60.465,-95.912,166.289,50.342,159.109
C05920=1021.406,-60.715,-95.902,166.285,50.347,159.109
C05921=1021.401,-60.964,-95.890,166.283,50.352,159.109
C05922=1021.395,-61.214,-95.879,166.280,50.356,159.110
C05923=1021.389,-61.463,-95.868,166.277,50.359,159.110
C05924=1021.383,-61.714,-95.858,166.273,50.363,159.110
C05925=1021.377,-61.964,-95.847,166.271,50.368,159.110
C05926=1021.372,-62.213,-95.836,166.268,50.372,159.110
C05927=1021.366,-62.463,-95.825,166.264,50.376,159.111
C05928=1021.360,-62.712,-95.814,166.262,50.380,159.111
C05929=1021.355,-62.962,-95.803,166.259,50.384,159.111
C05930=1021.350,-63.212,-95.792,166.255,50.389,159.111
C05931=1021.343,-63.462,-95.781,166.253,50.393,159.112
C05932=1021.338,-63.712,-95.771,166.250,50.397,159.112
C05933=1021.332,-63.961,-95.760,166.246,50.401,159.112
C05934=1021.326,-64.211,-95.749,166.244,50.405,159.112
C05935=1021.321,-64.460,-95.738,166.241,50.410,159.113
C05936=1021.315,-64.710,-95.727,166.238,50.414,159.113
C05937=1021.309,-64.959,-95.716,166.235,50.418,159.113
C05938=1021.304,-65.209,-95.706,166.232,50.422,159.113
C05939=1021.298,-65.459,-95.695,166.229,50.426,159.114
C05940=1021.293,-65.709,-95.684,166.226,50.431,159.114
C05941=1021.287,-65.958,-95.673,166.223,50.435,159.114
C05942=1021.282,-66.208,-95.663,166.220,50.438,159.114
C05943=1021.276,-66.458,-95.652,166.217,50.442,159.114
C05944=1021.270,-66.708,-95.640,166.213,50.447,159.115
C05945=1021.264,-66.957,-95.630,166.211,50.451,159.115
C05946=1021.258,-67.208,-95.619,166.208,50.455,159.115
C05947=1021.253,-67.457,-95.609,166.204,50.459,159.115
C05948=1021.247,-67.707,-95.598,166.202,50.463,159.116
C05949=1021.241,-67.956,-95.587,166.199,50.468,159.116
C05950=1021.236,-68.206,-95.577,166.196,50.472,159.116
C05951=1021.230,-68.456,-95.566,166.192,50.475,159.116
C05952=1021.225,-68.705,-95.554,166.190,50.480,159.116
C05953=1021.219,-68.986,-95.543,166.186,50.485,159.117
C05954=1021.213,-69.266,-95.531,166.184,50.489,159.117
C05955=1021.207,-69.547,-95.519,166.180,50.493,159.117
C05956=1021.201,-69.826,-95.507,166.177,50.498,159.117
C05957=1021.195,-70.076,-95.496,166.174,50.502,159.118
C05958=1021.189,-70.326,-95.486,166.170,50.506,159.118
C05959=1021.184,-70.576,-95.475,166.167,50.510,159.118
C05960=1021.178,-70.825,-95.464,166.165,50.514,159.118
C05961=1021.172,-71.075,-95.454,166.162,50.519,159.119
C05962=1021.167,-71.325,-95.443,166.158,50.522,159.119
C05963=1021.161,-71.575,-95.433,166.155,50.526,159.119
C05964=1021.156,-71.824,-95.422,166.153,50.530,159.119
C05965=1021.150,-72.074,-95.411,166.150,50.535,159.119
C05966=1021.144,-72.324,-95.401,166.146,50.539,159.120
C05967=1021.139,-72.573,-95.390,166.143,50.542,159.120
C05968=1021.133,-72.823,-95.380,166.140,50.547,159.120
C05969=1021.129,-73.073,-95.369,166.138,50.551,159.120
C05970=1021.123,-73.323,-95.359,166.134,50.555,159.120
C05971=1021.118,-73.572,-95.348,166.131,50.559,159.121
C05972=1021.112,-73.822,-95.338,166.128,50.563,159.121
C05973=1021.106,-74.072,-95.327,166.126,50.567,159.121
C05974=1021.101,-74.322,-95.317,166.122,50.571,159.121
C05975=1021.095,-74.571,-95.306,166.119,50.575,159.121
C05976=1021.090,-74.821,-95.296,166.117,50.579,159.122
C05977=1021.083,-75.071,-95.285,166.113,50.584,159.122
C05978=1021.079,-75.320,-95.276,166.110,50.588,159.122
C05979=1021.073,-75.570,-95.265,166.108,50.592,159.122
C05980=1021.067,-75.820,-95.254,166.104,50.597,159.123
C05981=1021.061,-76.069,-95.245,166.101,50.601,159.123
C05982=1021.056,-76.320,-95.235,166.098,50.604,159.123
C05983=1021.050,-76.569,-95.224,166.095,50.609,159.123
C05984=1021.045,-76.819,-95.214,166.092,50.613,159.123
C05985=1021.039,-77.068,-95.205,166.089,50.617,159.124
C05986=1021.033,-77.318,-95.194,166.086,50.621,159.124
C05987=1021.028,-77.568,-95.183,166.083,50.625,159.124
C05988=1021.022,-77.818,-95.173,166.080,50.629,159.124
C05989=1021.016,-78.068,-95.164,166.077,50.634,159.124
C05990=1021.011,-78.317,-95.153,166.074,50.638,159.125
C05991=1021.006,-78.567,-95.143,166.071,50.642,159.125
C05992=1021.000,-78.817,-95.133,166.068,50.647,159.125
C05993=1020.994,-79.067,-95.123,166.065,50.651,159.125
C05994=1020.988,-79.316,-95.112,166.062,50.654,159.126
C05995=1020.983,-79.565,-95.103,166.058,50.659,159.126
C05996=1020.978,-79.816,-95.093,166.056,50.663,159.126
C05997=1020.972,-80.065,-95.083,166.053,50.667,159.126
C05998=1020.966,-80.315,-95.073,166.049,50.671,159.126
C05999=1020.962,-80.565,-95.063,166.047,50.675,159.127
C06000=1020.955,-80.814,-95.053,166.043,50.680,159.127
C06001=1020.950,-81.064,-95.043,166.040,50.684,159.127
C06002=1020.944,-81.314,-95.033,166.038,50.688,159.127
C06003=1020.939,-81.563,-95.023,166.034,50.693,159.128
C06004=1020.933,-81.813,-95.014,166.031,50.697,159.128
C06005=1020.927,-82.063,-95.003,166.028,50.702,159.128
C06006=1020.921,-82.313,-94.994,166.025,50.706,159.128
C06007=1020.915,-82.562,-94.985,166.023,50.710,159.129
C06008=1020.910,-82.812,-94.975,166.019,50.715,159.129
C06009=1020.904,-83.062,-94.965,166.016,50.719,159.129
C06010=1020.898,-83.312,-94.955,166.013,50.723,159.129
C06011=1020.893,-83.561,-94.946,166.010,50.727,159.130
C06012=1020.887,-83.811,-94.935,166.007,50.732,159.130
C06013=1020.881,-84.061,-94.926,166.004,50.736,159.130
C06014=1020.876,-84.311,-94.916,166.001,50.740,159.130
C06015=1020.870,-84.560,-94.906,165.997,50.745,159.130
C06016=1020.865,-84.811,-94.896,165.995,50.749,159.131
C06017=1020.859,-85.093,-94.886,165.991,50.753,159.131
C06018=1020.852,-85.375,-94.875,165.988,50.758,159.131
C06019=1020.846,-85.657,-94.863,165.984,50.763,159.131
C06020=1020.840,-85.940,-94.853,165.981,50.768,159.132
C06021=1020.834,-86.189,-94.844,165.978,50.772,159.132
C06022=1020.829,-86.439,-94.833,165.974,50.777,159.132
C06023=1020.822,-86.689,-94.824,165.972,50.781,159.132
C06024=1020.818,-86.939,-94.814,165.969,50.785,159.133
C06025=1020.811,-87.188,-94.805,165.965,50.789,159.133
C06026=1020.806,-87.439,-94.796,165.963,50.794,159.133
C06027=1020.801,-87.688,-94.786,165.959,50.798,159.133
C06028=1020.795,-87.938,-94.776,165.956,50.802,159.133
C06029=1020.790,-88.187,-94.767,165.953,50.806,159.133
C06030=1020.784,-88.437,-94.757,165.950,50.810,159.134
C06031=1020.778,-88.687,-94.747,165.947,50.814,159.134
C06032=1020.773,-88.936,-94.738,165.944,50.818,159.134
C06033=1020.767,-89.187,-94.728,165.941,50.823,159.134
C06034=1020.762,-89.436,-94.719,165.938,50.827,159.135
C06035=1020.756,-89.686,-94.709,165.935,50.831,159.135
C06036=1020.751,-89.935,-94.700,165.932,50.836,159.135
C06037=1020.745,-90.185,-94.690,165.929,50.840,159.135
C06038=1020.740,-90.435,-94.681,165.925,50.844,159.135
C06039=1020.734,-90.685,-94.671,165.923,50.848,159.136
C06040=1020.729,-90.934,-94.662,165.920,50.852,159.136
C06041=1020.723,-91.184,-94.652,165.916,50.856,159.136
C06042=1020.718,-91.434,-94.643,165.913,50.860,159.136
C06043=1020.712,-91.684,-94.633,165.911,50.865,159.136
C06044=1020.707,-91.933,-94.624,165.907,50.869,159.137
C06045=1020.702,-92.184,-94.615,165.904,50.873,159.137
C06046=1020.696,-92.433,-94.606,165.902,50.877,159.137
C06047=1020.691,-92.683,-94.595,165.898,50.882,159.137
C06048=1020.685,-92.932,-94.586,165.895,50.886,159.138
C06049=1020.680,-93.183,-94.577,165.892,50.889,159.138
C06050=1020.674,-93.432,-94.568,165.889,50.894,159.138
C06051=1020.669,-93.682,-94.557,165.886,50.898,159.138
C06052=1020.664,-93.932,-94.549,165.883,50.902,159.138
C06053=1020.657,-94.182,-94.539,165.880,50.907,159.138
C06054=1020.653,-94.431,-94.530,165.877,50.911,159.139
C06055=1020.647,-94.681,-94.521,165.874,50.914,159.139
C06056=1020.642,-94.931,-94.511,165.870,50.919,159.139
C06057=1020.637,-95.181,-94.502,165.868,50.923,159.139
C06058=1020.631,-95.431,-94.492,165.865,50.927,159.139
C06059=1020.626,-95.680,-94.483,165.861,50.932,159.140
C06060=1020.620,-95.930,-94.474,165.858,50.935,159.140
C06061=1020.615,-96.180,-94.464,165.856,50.939,159.140
C06062=1020.609,-96.430,-94.456,165.852,50.944,159.140
C06063=1020.604,-96.679,-94.446,165.849,50.948,159.140
C06064=1020.599,-96.929,-94.437,165.847,50.952,159.141
C06065=1020.593,-97.179,-94.428,165.843,50.956,159.140
C06066=1020.588,-97.428,-94.418,165.840,50.960,159.141
C06067=1020.582,-97.679,-94.409,165.838,50.964,159.141
C06068=1020.577,-97.928,-94.399,165.834,50.969,159.141
C06069=1020.572,-98.178,-94.391,165.831,50.973,159.141
C06070=1020.566,-98.428,-94.382,165.829,50.977,159.142
C06071=1020.561,-98.677,-94.373,165.825,50.981,159.142
C06072=1020.555,-98.927,-94.364,165.822,50.986,159.142
C06073=1020.549,-99.177,-94.355,165.819,50.990,159.142
C06074=1020.545,-99.427,-94.346,165.816,50.994,159.142
C06075=1020.539,-99.677,-94.337,165.813,50.998,159.143
C06076=1020.533,-99.926,-94.328,165.810,51.003,159.143
C06077=1020.528,-100.176,-94.319,165.807,51.007,159.143
C06078=1020.523,-100.426,-94.311,165.803,51.011,159.143
C06079=1020.516,-100.676,-94.301,165.800,51.015,159.143
C06080=1020.511,-100.925,-94.292,165.798,51.019,159.144
C06081=1020.505,-101.210,-94.282,165.794,51.024,159.144
C06082=1020.499,-101.495,-94.272,165.791,51.029,159.144
C06083=1020.493,-101.779,-94.262,165.787,51.034,159.144
C06084=1020.486,-102.063,-94.252,165.784,51.039,159.145
C06085=1020.482,-102.313,-94.243,165.780,51.043,159.145
C06086=1020.476,-102.563,-94.234,165.777,51.047,159.145
C06087=1020.470,-102.814,-94.225,165.775,51.051,159.145
C06088=1020.465,-103.063,-94.216,165.771,51.056,159.145
C06089=1020.460,-103.312,-94.207,165.768,51.060,159.146
C06090=1020.454,-103.562,-94.199,165.765,51.065,159.146
C06091=1020.448,-103.812,-94.190,165.762,51.069,159.146
C06092=1020.443,-104.062,-94.181,165.759,51.072,159.146
C06093=1020.438,-104.312,-94.172,165.756,51.077,159.146
C06094=1020.433,-104.561,-94.163,165.753,51.081,159.146
C06095=1020.427,-104.812,-94.155,165.750,51.085,159.147
C06096=1020.422,-105.061,-94.146,165.747,51.089,159.147
C06097=1020.416,-105.311,-94.137,165.744,51.094,159.147
C06098=1020.411,-105.560,-94.128,165.741,51.098,159.147
C06099=1020.406,-105.810,-94.120,165.738,51.102,159.147
C06100=1020.400,-106.060,-94.111,165.735,51.106,159.148
C06101=1020.395,-106.310,-94.103,165.731,51.110,159.148
C06102=1020.389,-106.560,-94.094,165.728,51.114,159.148
C06103=1020.384,-106.810,-94.086,165.726,51.119,159.148
C06104=1020.379,-107.059,-94.077,165.722,51.123,159.148
C06105=1020.373,-107.309,-94.068,165.719,51.127,159.149
C06106=1020.367,-107.559,-94.059,165.717,51.132,159.149
C06107=1020.363,-107.809,-94.050,165.713,51.136,159.149
C06108=1020.357,-108.058,-94.042,165.710,51.140,159.149
C06109=1020.352,-108.308,-94.034,165.707,51.145,159.149
C06110=1020.346,-108.558,-94.025,165.704,51.149,159.150
C06111=1020.341,-108.808,-94.016,165.701,51.152,159.150
C06112=1020.335,-109.058,-94.008,165.697,51.157,159.150
C06113=1020.330,-109.307,-93.999,165.695,51.161,159.150
C06114=1020.325,-109.557,-93.991,165.691,51.166,159.150
C06115=1020.319,-109.807,-93.982,165.689,51.170,159.150
C06116=1020.314,-110.057,-93.974,165.686,51.174,159.151
C06117=1020.309,-110.306,-93.965,165.682,51.178,159.151
C06118=1020.304,-110.557,-93.958,165.680,51.183,159.151
C06119=1020.299,-110.806,-93.949,165.677,51.187,159.151
C06120=1020.292,-111.056,-93.941,165.673,51.191,159.151
C06121=1020.287,-111.306,-93.932,165.671,51.196,159.152
C06122=1020.282,-111.556,-93.924,165.667,51.200,159.152
C06123=1020.276,-111.806,-93.915,165.664,51.204,159.152
C06124=1020.271,-112.055,-93.907,165.661,51.208,159.152
C06125=1020.266,-112.305,-93.898,165.658,51.212,159.152
C06126=1020.261,-112.555,-93.890,165.655,51.216,159.153
C06127=1020.255,-112.804,-93.881,165.653,51.221,159.153
C06128=1020.250,-113.055,-93.874,165.649,51.225,159.153
C06129=1020.245,-113.305,-93.865,165.646,51.229,159.153
C06130=1020.239,-113.554,-93.857,165.643,51.234,159.153
C06131=1020.234,-113.804,-93.849,165.640,51.238,159.154
C06132=1020.229,-114.053,-93.840,165.637,51.242,159.154
C06133=1020.223,-114.303,-93.832,165.633,51.246,159.154
C06134=1020.218,-114.553,-93.824,165.631,51.250,159.154
C06135=1020.213,-114.803,-93.816,165.628,51.254,159.154
C06136=1020.208,-115.053,-93.807,165.624,51.259,159.154
C06137=1020.202,-115.302,-93.799,165.622,51.263,159.155
C06138=1020.197,-115.553,-93.791,165.618,51.268,159.155
C06139=1020.192,-115.802,-93.783,165.615,51.272,159.155
C06140=1020.186,-116.052,-93.774,165.613,51.276,159.155
C06141=1020.180,-116.301,-93.767,165.609,51.281,159.155
C06142=1020.175,-116.552,-93.759,165.607,51.285,159.156
C06143=1020.170,-116.801,-93.750,165.604,51.289,159.156
C06144=1020.165,-117.051,-93.742,165.600,51.293,159.156
C06145=1020.159,-117.335,-93.733,165.597,51.298,159.156
C06146=1020.152,-117.620,-93.724,165.593,51.303,159.156
C06147=1020.146,-117.904,-93.715,165.590,51.308,159.157
C06148=1020.140,-118.189,-93.705,165.586,51.312,159.157
C06149=1020.135,-118.439,-93.697,165.583,51.316,159.157
C06150=1020.130,-118.688,-93.690,165.581,51.321,159.157
C06151=1020.125,-118.938,-93.682,165.577,51.325,159.157
C06152=1020.120,-119.188,-93.673,165.575,51.329,159.158
C06153=1020.114,-119.437,-93.666,165.571,51.334,159.158
C06154=1020.109,-119.688,-93.658,165.568,51.338,159.158
C06155=1020.103,-119.937,-93.649,165.566,51.342,159.158
C06156=1020.098,-120.188,-93.642,165.562,51.347,159.158
C06157=1020.092,-120.437,-93.634,165.559,51.350,159.158
C06158=1020.088,-120.688,-93.626,165.556,51.355,159.159
C06159=1020.083,-120.937,-93.618,165.553,51.359,159.159
C06160=1020.077,-121.187,-93.611,165.550,51.363,159.159
C06161=1020.072,-121.436,-93.602,165.547,51.368,159.159
C06162=1020.067,-121.687,-93.594,165.544,51.372,159.159
C06163=1020.061,-121.936,-93.586,165.541,51.376,159.160
C06164=1020.056,-122.186,-93.579,165.538,51.381,159.160
C06165=1020.051,-122.436,-93.570,165.535,51.385,159.160
C06166=1020.046,-122.685,-93.563,165.532,51.388,159.160
C06167=1020.040,-122.935,-93.555,165.528,51.393,159.160
C06168=1020.035,-123.185,-93.547,165.526,51.397,159.160
C06169=1020.029,-123.435,-93.539,165.523,51.401,159.161
C06170=1020.024,-123.685,-93.531,165.519,51.406,159.161
C06171=1020.020,-123.934,-93.523,165.517,51.410,159.161
C06172=1020.014,-124.184,-93.516,165.514,51.414,159.161
C06173=1020.009,-124.435,-93.508,165.510,51.418,159.161
C06174=1020.004,-124.684,-93.500,165.507,51.422,159.161
C06175=1019.998,-124.934,-93.493,165.505,51.427,159.162
C06176=1019.994,-125.184,-93.485,165.501,51.431,159.162
C06177=1019.988,-125.433,-93.477,165.499,51.435,159.162
C06178=1019.983,-125.684,-93.470,165.495,51.440,159.162
C06179=1019.977,-125.934,-93.462,165.492,51.444,159.162
C06180=1019.972,-126.183,-93.454,165.490,51.448,159.163
C06181=1019.967,-126.433,-93.447,165.486,51.453,159.163
C06182=1019.962,-126.683,-93.439,165.483,51.457,159.163
C06183=1019.956,-126.932,-93.432,165.481,51.461,159.163
C06184=1019.951,-127.182,-93.424,165.477,51.466,159.163
C06185=1019.946,-127.432,-93.417,165.475,51.470,159.164
C06186=1019.940,-127.682,-93.408,165.472,51.474,159.164
C06187=1019.935,-127.931,-93.402,165.468,51.478,159.164
C06188=1019.930,-128.182,-93.394,165.465,51.482,159.164
C06189=1019.926,-128.431,-93.386,165.462,51.486,159.164
C06190=1019.921,-128.681,-93.377,165.459,51.489,159.164
C06191=1019.918,-128.930,-93.367,165.457,51.492,159.164
C06192=1019.915,-129.180,-93.357,165.454,51.493,159.164
C06193=1019.912,-129.430,-93.346,165.451,51.495,159.164
C06194=1019.910,-129.679,-93.335,165.449,51.496,159.163
C06195=1019.908,-129.928,-93.323,165.446,51.497,159.163
C06196=1019.906,-130.178,-93.311,165.444,51.497,159.162
C06197=1019.905,-130.428,-93.298,165.442,51.496,159.162
C06198=1019.905,-130.678,-93.284,165.439,51.495,159.161
C06199=1019.905,-130.927,-93.270,165.437,51.493,159.160
C06200=1019.905,-131.177,-93.255,165.435,51.491,159.160
C06201=1019.906,-131.427,-93.239,165.433,51.488,159.159
C06202=1019.907,-131.677,-93.223,165.431,51.485,159.158
C06203=1019.909,-131.927,-93.207,165.429,51.482,159.157
C06204=1019.912,-132.176,-93.190,165.427,51.477,159.156
C06205=1019.914,-132.426,-93.172,165.426,51.473,159.155
C06206=1019.917,-132.676,-93.154,165.424,51.468,159.154
C06207=1019.921,-132.925,-93.135,165.422,51.462,159.152
C06208=1019.924,-133.175,-93.115,165.420,51.456,159.151
C06209=1019.649,-133.201,-93.479,165.377,51.769,159.197
C06210=1019.646,-132.952,-93.499,165.378,51.775,159.198
C06211=1019.642,-132.702,-93.518,165.380,51.781,159.199
C06212=1019.639,-132.452,-93.537,165.381,51.786,159.200
C06213=1019.637,-132.202,-93.554,165.384,51.791,159.202
C06214=1019.634,-131.953,-93.571,165.385,51.795,159.203
C06215=1019.632,-131.703,-93.588,165.387,51.798,159.204
C06216=1019.631,-131.453,-93.604,165.389,51.802,159.205
C06217=1019.630,-131.203,-93.619,165.392,51.805,159.205
C06218=1019.630,-130.954,-93.634,165.394,51.806,159.206
C06219=1019.630,-130.704,-93.648,165.396,51.808,159.207
C06220=1019.630,-130.454,-93.662,165.398,51.809,159.208
C06221=1019.631,-130.204,-93.675,165.400,51.810,159.208
C06222=1019.632,-129.955,-93.687,165.403,51.810,159.208
C06223=1019.634,-129.705,-93.699,165.405,51.809,159.209
C06224=1019.637,-129.455,-93.710,165.407,51.808,159.209
C06225=1019.640,-129.205,-93.721,165.410,51.807,159.209
C06226=1019.643,-128.956,-93.731,165.413,51.805,159.209
C06227=1019.646,-128.706,-93.741,165.416,51.802,159.210
C06228=1019.650,-128.456,-93.750,165.418,51.799,159.209
C06229=1019.655,-128.207,-93.758,165.421,51.795,159.209
C06230=1019.660,-127.958,-93.766,165.425,51.791,159.209
C06231=1019.665,-127.708,-93.773,165.428,51.787,159.209
C06232=1019.670,-127.458,-93.781,165.430,51.783,159.209
C06233=1019.676,-127.209,-93.789,165.434,51.778,159.209
C06234=1019.681,-126.959,-93.796,165.436,51.774,159.209
C06235=1019.686,-126.709,-93.804,165.439,51.770,159.208
C06236=1019.691,-126.459,-93.811,165.443,51.765,159.208
C06237=1019.697,-126.210,-93.819,165.445,51.761,159.208
C06238=1019.702,-125.960,-93.827,165.449,51.757,159.208
C06239=1019.707,-125.710,-93.834,165.451,51.752,159.208
C06240=1019.712,-125.459,-93.842,165.455,51.748,159.208
C06241=1019.718,-125.211,-93.849,165.458,51.743,159.207
C06242=1019.723,-124.960,-93.857,165.460,51.739,159.207
C06243=1019.728,-124.710,-93.865,165.464,51.735,159.207
C06244=1019.734,-124.461,-93.872,165.466,51.730,159.207
C06245=1019.738,-124.211,-93.880,165.470,51.727,159.207
C06246=1019.744,-123.961,-93.887,165.473,51.722,159.207
C06247=1019.749,-123.711,-93.896,165.476,51.718,159.206
C06248=1019.754,-123.461,-93.903,165.479,51.714,159.206
C06249=1019.760,-123.211,-93.911,165.482,51.709,159.206
C06250=1019.764,-122.962,-93.919,165.484,51.705,159.206
C06251=1019.769,-122.711,-93.926,165.488,51.700,159.206
C06252=1019.775,-122.462,-93.934,165.491,51.696,159.205
C06253=1019.780,-122.212,-93.942,165.494,51.692,159.205
C06254=1019.785,-121.962,-93.951,165.497,51.687,159.205
C06255=1019.791,-121.713,-93.957,165.499,51.683,159.205
C06256=1019.796,-121.463,-93.966,165.503,51.679,159.205
C06257=1019.801,-121.213,-93.974,165.506,51.675,159.205
C06258=1019.807,-120.963,-93.981,165.510,51.671,159.204
C06259=1019.812,-120.713,-93.989,165.512,51.666,159.204
C06260=1019.817,-120.463,-93.998,165.515,51.662,159.204
C06261=1019.821,-120.214,-94.005,165.518,51.658,159.204
C06262=1019.827,-119.964,-94.013,165.521,51.653,159.204
C06263=1019.832,-119.714,-94.021,165.524,51.649,159.203
C06264=1019.838,-119.464,-94.029,165.527,51.645,159.203
C06265=1019.843,-119.214,-94.036,165.530,51.640,159.203
C06266=1019.849,-118.964,-94.045,165.533,51.636,159.203
C06267=1019.854,-118.715,-94.053,165.536,51.632,159.203
C06268=1019.860,-118.465,-94.061,165.540,51.627,159.203
C06269=1019.864,-118.216,-94.069,165.542,51.623,159.202
C06270=1019.870,-117.931,-94.078,165.546,51.618,159.202
C06271=1019.876,-117.647,-94.087,165.549,51.613,159.202
C06272=1019.882,-117.363,-94.096,165.553,51.608,159.202
C06273=1019.889,-117.078,-94.106,165.556,51.603,159.201
C06274=1019.894,-116.828,-94.113,165.559,51.599,159.201
C06275=1019.899,-116.578,-94.122,165.562,51.594,159.201
C06276=1019.904,-116.329,-94.130,165.565,51.591,159.201
C06277=1019.909,-116.079,-94.137,165.569,51.586,159.201
C06278=1019.915,-115.829,-94.146,165.571,51.582,159.201
C06279=1019.920,-115.579,-94.154,165.574,51.578,159.200
C06280=1019.925,-115.330,-94.163,165.578,51.573,159.200
C06281=1019.931,-115.080,-94.170,165.580,51.569,159.200
C06282=1019.936,-114.830,-94.178,165.584,51.564,159.200
C06283=1019.941,-114.580,-94.187,165.586,51.560,159.200
C06284=1019.946,-114.330,-94.194,165.590,51.556,159.199
C06285=1019.952,-114.080,-94.203,165.593,51.551,159.199
C06286=1019.957,-113.830,-94.211,165.595,51.547,159.199
C06287=1019.962,-113.581,-94.220,165.599,51.543,159.199
C06288=1019.968,-113.331,-94.228,165.602,51.538,159.199
C06289=1019.973,-113.081,-94.236,165.605,51.534,159.198
C06290=1019.978,-112.831,-94.244,165.608,51.530,159.198
C06291=1019.984,-112.582,-94.253,165.610,51.525,159.198
C06292=1019.989,-112.332,-94.261,165.614,51.521,159.198
C06293=1019.994,-112.082,-94.270,165.617,51.517,159.198
C06294=1019.999,-111.832,-94.278,165.621,51.513,159.198
C06295=1020.005,-111.583,-94.286,165.623,51.509,159.197
C06296=1020.010,-111.332,-94.294,165.626,51.504,159.197
C06297=1020.016,-111.082,-94.303,165.629,51.500,159.197
C06298=1020.021,-110.833,-94.311,165.632,51.496,159.197
C06299=1020.027,-110.583,-94.319,165.636,51.491,159.197
C06300=1020.032,-110.333,-94.328,165.638,51.487,159.196
C06301=1020.037,-110.083,-94.336,165.642,51.482,159.196
C06302=1020.043,-109.834,-94.345,165.645,51.478,159.196
C06303=1020.048,-109.584,-94.353,165.647,51.474,159.196
C06304=1020.053,-109.334,-94.362,165.651,51.469,159.196
C06305=1020.058,-109.085,-94.370,165.653,51.465,159.195
C06306=1020.064,-108.835,-94.379,165.657,51.461,159.195
C06307=1020.069,-108.585,-94.387,165.660,51.456,159.195
C06308=1020.075,-108.335,-94.396,165.663,51.452,159.195
C06309=1020.081,-108.085,-94.404,165.666,51.448,159.195
C06310=1020.086,-107.836,-94.413,165.668,51.444,159.194
C06311=1020.091,-107.586,-94.421,165.672,51.439,159.194
C06312=1020.097,-107.336,-94.430,165.675,51.435,159.194
C06313=1020.102,-107.086,-94.438,165.678,51.430,159.194
C06314=1020.106,-106.836,-94.447,165.681,51.426,159.194
C06315=1020.112,-106.586,-94.456,165.684,51.422,159.193
C06316=1020.117,-106.336,-94.464,165.687,51.417,159.193
C06317=1020.123,-106.087,-94.473,165.690,51.413,159.193
C06318=1020.128,-105.837,-94.481,165.694,51.409,159.193
C06319=1020.133,-105.587,-94.490,165.696,51.405,159.193
C06320=1020.138,-105.337,-94.498,165.699,51.401,159.193
C06321=1020.144,-105.087,-94.507,165.703,51.396,159.192
C06322=1020.150,-104.838,-94.516,165.705,51.392,159.192
C06323=1020.155,-104.588,-94.525,165.709,51.388,159.192
C06324=1020.160,-104.338,-94.533,165.711,51.383,159.192
C06325=1020.166,-104.089,-94.542,165.714,51.379,159.191
C06326=1020.172,-103.838,-94.551,165.718,51.375,159.191
C06327=1020.176,-103.589,-94.561,165.720,51.370,159.191
C06328=1020.182,-103.339,-94.569,165.724,51.366,159.191
C06329=1020.187,-103.089,-94.578,165.727,51.362,159.191
C06330=1020.193,-102.839,-94.586,165.730,51.357,159.191
C06331=1020.198,-102.589,-94.595,165.733,51.353,159.190
C06332=1020.204,-102.340,-94.604,165.735,51.349,159.190
C06333=1020.209,-102.091,-94.613,165.739,51.344,159.190
C06334=1020.215,-101.806,-94.623,165.743,51.340,159.190
C06335=1020.221,-101.521,-94.633,165.746,51.335,159.189
C06336=1020.228,-101.237,-94.643,165.750,51.330,159.189
C06337=1020.234,-100.953,-94.653,165.753,51.325,159.189
C06338=1020.239,-100.703,-94.662,165.756,51.321,159.189
C06339=1020.244,-100.453,-94.671,165.759,51.316,159.189
C06340=1020.249,-100.203,-94.680,165.762,51.312,159.188
C06341=1020.255,-99.953,-94.689,165.765,51.307,159.188
C06342=1020.261,-99.704,-94.698,165.768,51.303,159.188
C06343=1020.266,-99.454,-94.706,165.772,51.299,159.188
C06344=1020.272,-99.204,-94.716,165.774,51.294,159.188
C06345=1020.277,-98.954,-94.724,165.777,51.290,159.187
C06346=1020.282,-98.704,-94.733,165.781,51.286,159.187
C06347=1020.288,-98.455,-94.743,165.783,51.282,159.187
C06348=1020.293,-98.205,-94.751,165.787,51.277,159.187
C06349=1020.299,-97.956,-94.760,165.789,51.273,159.187
C06350=1020.305,-97.705,-94.769,165.793,51.268,159.186
C06351=1020.310,-97.456,-94.779,165.796,51.264,159.186
C06352=1020.315,-97.206,-94.788,165.799,51.261,159.186
C06353=1020.320,-96.955,-94.797,165.802,51.256,159.186
C06354=1020.325,-96.706,-94.806,165.805,51.252,159.186
C06355=1020.332,-96.457,-94.816,165.808,51.248,159.185
C06356=1020.336,-96.207,-94.825,165.811,51.243,159.185
C06357=1020.342,-95.957,-94.834,165.814,51.239,159.185
C06358=1020.347,-95.707,-94.844,165.817,51.236,159.185
C06359=1020.352,-95.458,-94.853,165.820,51.231,159.185
C06360=1020.358,-95.207,-94.862,165.823,51.227,159.185
C06361=1020.363,-94.958,-94.871,165.827,51.222,159.184
C06362=1020.369,-94.709,-94.881,165.829,51.218,159.184
C06363=1020.374,-94.458,-94.890,165.832,51.214,159.184
C06364=1020.379,-94.209,-94.899,165.836,51.209,159.184
C06365=1020.385,-93.958,-94.909,165.838,51.205,159.183
C06366=1020.390,-93.709,-94.918,165.841,51.201,159.183
C06367=1020.396,-93.459,-94.927,165.845,51.197,159.183
C06368=1020.401,-93.209,-94.936,165.847,51.193,159.183
C06369=1020.406,-92.960,-94.946,165.851,51.189,159.183
C06370=1020.412,-92.710,-94.956,165.854,51.184,159.183
C06371=1020.417,-92.460,-94.964,165.856,51.180,159.182
C06372=1020.423,-92.210,-94.975,165.860,51.176,159.182
C06373=1020.428,-91.961,-94.984,165.863,51.172,159.182
C06374=1020.434,-91.711,-94.993,165.865,51.167,159.182
C06375=1020.439,-91.461,-95.002,165.869,51.163,159.182
C06376=1020.445,-91.212,-95.012,165.872,51.159,159.181
C06377=1020.449,-90.961,-95.021,165.875,51.154,159.181
C06378=1020.456,-90.712,-95.031,165.878,51.150,159.181
C06379=1020.460,-90.462,-95.040,165.880,51.146,159.181
C06380=1020.467,-90.212,-95.050,165.884,51.141,159.180
C06381=1020.472,-89.963,-95.058,165.887,51.137,159.180
C06382=1020.477,-89.713,-95.069,165.891,51.133,159.180
C06383=1020.483,-89.464,-95.078,165.893,51.129,159.180
C06384=1020.488,-89.213,-95.088,165.896,51.125,159.180
C06385=1020.494,-88.964,-95.097,165.900,51.121,159.180
C06386=1020.499,-88.714,-95.107,165.902,51.116,159.179
C06387=1020.505,-88.464,-95.116,165.906,51.112,159.179
C06388=1020.510,-88.214,-95.126,165.909,51.108,159.179
C06389=1020.516,-87.965,-95.136,165.912,51.103,159.179
C06390=1020.521,-87.715,-95.145,165.915,51.099,159.178
C06391=1020.527,-87.465,-95.154,165.917,51.095,159.178
C06392=1020.533,-87.216,-95.163,165.921,51.090,159.178
C06393=1020.538,-86.966,-95.174,165.924,51.086,159.178
C06394=1020.544,-86.716,-95.183,165.927,51.082,159.178
C06395=1020.549,-86.466,-95.193,165.930,51.077,159.177
C06396=1020.555,-86.217,-95.202,165.933,51.072,159.177
C06397=1020.560,-85.967,-95.212,165.936,51.068,159.177
C06398=1020.566,-85.684,-95.223,165.940,51.064,159.177
C06399=1020.573,-85.402,-95.234,165.943,51.058,159.176
C06400=1020.578,-85.120,-95.244,165.946,51.054,159.176
C06401=1020.585,-84.838,-95.256,165.950,51.049,159.176
C06402=1020.591,-84.588,-95.265,165.952,51.045,159.176
C06403=1020.597,-84.339,-95.275,165.956,51.040,159.175
C06404=1020.602,-84.089,-95.285,165.959,51.036,159.175
C06405=1020.608,-83.839,-95.294,165.962,51.031,159.175
C06406=1020.613,-83.589,-95.304,165.965,51.027,159.175
C06407=1020.619,-83.340,-95.314,165.969,51.023,159.175
C06408=1020.625,-83.089,-95.324,165.971,51.019,159.174
C06409=1020.630,-82.840,-95.333,165.975,51.013,159.174
C06410=1020.636,-82.590,-95.343,165.977,51.009,159.174
C06411=1020.642,-82.340,-95.353,165.980,51.005,159.173
C06412=1020.647,-82.090,-95.363,165.983,51.001,159.173
C06413=1020.653,-81.841,-95.372,165.986,50.996,159.173
C06414=1020.658,-81.591,-95.382,165.990,50.992,159.173
C06415=1020.665,-81.341,-95.392,165.992,50.988,159.173
C06416=1020.669,-81.092,-95.402,165.996,50.983,159.172
C06417=1020.676,-80.842,-95.411,165.999,50.979,159.172
C06418=1020.681,-80.592,-95.421,166.002,50.974,159.172
C06419=1020.687,-80.342,-95.431,166.005,50.970,159.171
C06420=1020.692,-80.093,-95.441,166.008,50.965,159.171
C06421=1020.697,-79.843,-95.451,166.011,50.961,159.171
C06422=1020.704,-79.593,-95.460,166.013,50.957,159.171
C06423=1020.709,-79.343,-95.471,166.017,50.952,159.171
C06424=1020.714,-79.094,-95.481,166.020,50.948,159.170
C06425=1020.720,-78.844,-95.491,166.022,50.944,159.170
C06426=1020.726,-78.594,-95.501,166.026,50.940,159.170
C06427=1020.731,-78.344,-95.511,166.029,50.936,159.170
C06428=1020.737,-78.094,-95.521,166.033,50.932,159.170
C06429=1020.743,-77.845,-95.531,166.035,50.928,159.169
C06430=1020.748,-77.595,-95.541,166.038,50.923,159.169
C06431=1020.753,-77.345,-95.551,166.042,50.919,159.169
C06432=1020.759,-77.096,-95.562,166.044,50.915,159.169
C06433=1020.764,-76.846,-95.572,166.047,50.911,159.168
C06434=1020.770,-76.596,-95.582,166.051,50.906,159.168
C06435=1020.776,-76.346,-95.592,166.053,50.902,159.168
C06436=1020.781,-76.097,-95.603,166.057,50.898,159.168
C06437=1020.787,-75.847,-95.613,166.060,50.893,159.168
C06438=1020.793,-75.597,-95.622,166.062,50.889,159.167
C06439=1020.798,-75.348,-95.633,166.066,50.885,159.167
C06440=1020.804,-75.098,-95.643,166.068,50.880,159.167
C06441=1020.809,-74.848,-95.653,166.072,50.875,159.167
C06442=1020.815,-74.599,-95.663,166.074,50.871,159.166
C06443=1020.821,-74.349,-95.674,166.077,50.867,159.166
C06444=1020.826,-74.099,-95.684,166.081,50.863,159.166
C06445=1020.832,-73.849,-95.695,166.084,50.859,159.166
C06446=1020.837,-73.599,-95.705,166.086,50.855,159.165
C06447=1020.843,-73.350,-95.715,166.090,50.851,159.165
C06448=1020.847,-73.100,-95.726,166.093,50.847,159.165
C06449=1020.853,-72.850,-95.737,166.095,50.842,159.165
C06450=1020.858,-72.600,-95.747,166.098,50.839,159.165
C06451=1020.864,-72.351,-95.758,166.102,50.834,159.165
C06452=1020.870,-72.101,-95.769,166.105,50.830,159.164
C06453=1020.875,-71.851,-95.779,166.107,50.826,159.164
C06454=1020.881,-71.602,-95.790,166.111,50.822,159.164
C06455=1020.886,-71.352,-95.800,166.114,50.818,159.164
C06456=1020.892,-71.103,-95.811,166.116,50.813,159.163
C06457=1020.897,-70.853,-95.821,166.120,50.809,159.163
C06458=1020.903,-70.603,-95.832,166.123,50.806,159.163
C06459=1020.909,-70.354,-95.843,166.125,50.801,159.163
C06460=1020.914,-70.103,-95.853,166.129,50.797,159.163
C06461=1020.920,-69.854,-95.864,166.132,50.793,159.162
C06462=1020.926,-69.573,-95.875,166.135,50.788,159.162
C06463=1020.932,-69.293,-95.887,166.139,50.783,159.162
C06464=1020.939,-69.013,-95.900,166.141,50.779,159.162
C06465=1020.944,-68.733,-95.911,166.145,50.774,159.161
C06466=1020.950,-68.483,-95.922,166.148,50.769,159.161
C06467=1020.956,-68.233,-95.932,166.151,50.765,159.161
C06468=1020.961,-67.984,-95.943,166.154,50.761,159.160
C06469=1020.966,-67.734,-95.954,166.157,50.757,159.160
C06470=1020.972,-67.485,-95.965,166.160,50.753,159.160
C06471=1020.977,-67.234,-95.975,166.163,50.749,159.160
C06472=1020.983,-66.985,-95.986,166.167,50.745,159.160
C06473=1020.989,-66.735,-95.997,166.169,50.741,159.159
C06474=1020.994,-66.485,-96.007,166.172,50.736,159.159
C06475=1021.000,-66.236,-96.018,166.176,50.732,159.159
C06476=1021.006,-65.986,-96.029,166.178,50.728,159.159
C06477=1021.012,-65.737,-96.040,166.181,50.724,159.158
C06478=1021.017,-65.487,-96.050,166.185,50.719,159.158
C06479=1021.022,-65.237,-96.062,166.187,50.715,159.158
C06480=1021.028,-64.987,-96.072,166.190,50.711,159.158
C06481=1021.034,-64.737,-96.084,166.194,50.707,159.158
C06482=1021.039,-64.487,-96.094,166.196,50.702,159.157
C06483=1021.045,-64.238,-96.105,166.199,50.698,159.157
C06484=1021.051,-63.988,-96.116,166.203,50.694,159.157
C06485=1021.057,-63.739,-96.126,166.205,50.690,159.157
C06486=1021.062,-63.489,-96.137,166.208,50.686,159.156
C06487=1021.068,-63.239,-96.148,166.211,50.681,159.156
C06488=1021.074,-62.990,-96.158,166.214,50.677,159.156
C06489=1021.079,-62.740,-96.169,166.217,50.673,159.156
C06490=1021.084,-62.490,-96.181,166.220,50.668,159.155
C06491=1021.090,-62.241,-96.192,166.223,50.664,159.155
C06492=1021.096,-61.991,-96.203,166.225,50.659,159.155
C06493=1021.102,-61.741,-96.214,166.229,50.655,159.154
C06494=1021.108,-61.491,-96.224,166.232,50.651,159.154
C06495=1021.113,-61.242,-96.235,166.235,50.646,159.154
C06496=1021.119,-60.992,-96.246,166.238,50.642,159.154
C06497=1021.125,-60.743,-96.257,166.241,50.638,159.153
C06498=1021.131,-60.493,-96.267,166.244,50.634,159.153
C06499=1021.136,-60.243,-96.279,166.247,50.630,159.153
C06500=1021.142,-59.993,-96.290,166.250,50.625,159.153
C06501=1021.148,-59.744,-96.301,166.253,50.621,159.153
C06502=1021.153,-59.494,-96.312,166.256,50.617,159.152
C06503=1021.159,-59.245,-96.323,166.258,50.612,159.152
C06504=1021.165,-58.995,-96.334,166.262,50.608,159.152
///RCONF 1,0,0,0,0,0,0,0,0,0,0,0,0,0,0,0,0,0,0,0,0,0,0,0
C06505=1021.171,-58.745,-96.345,166.265,50.604,159.151
C06506=1021.177,-58.495,-96.356,166.268,50.599,159.151
C06507=1021.182,-58.245,-96.367,166.271,50.595,159.151
C06508=1021.187,-57.996,-96.377,166.274,50.591,159.151
C06509=1021.193,-57.746,-96.388,166.277,50.586,159.150
C06510=1021.199,-57.496,-96.400,166.280,50.582,159.150
C06511=1021.205,-57.246,-96.410,166.283,50.577,159.150
C06512=1021.211,-56.998,-96.422,166.286,50.573,159.150
C06513=1021.217,-56.748,-96.433,166.288,50.569,159.149
C06514=1021.223,-56.498,-96.444,166.292,50.564,159.149
C06515=1021.228,-56.248,-96.456,166.295,50.560,159.149
C06516=1021.234,-55.999,-96.466,166.297,50.556,159.148
C06517=1021.240,-55.749,-96.477,166.301,50.551,159.148
C06518=1021.246,-55.499,-96.489,166.303,50.547,159.148
C06519=1021.252,-55.249,-96.499,166.307,50.543,159.148
C06520=1021.258,-55.000,-96.510,166.310,50.538,159.147
C06521=1021.264,-54.750,-96.522,166.312,50.534,159.147
C06522=1021.269,-54.500,-96.533,166.316,50.529,159.147
C06523=1021.275,-54.250,-96.544,166.318,50.525,159.146
C06524=1021.280,-54.001,-96.555,166.322,50.521,159.146
C06525=1021.287,-53.751,-96.566,166.325,50.517,159.146
C06526=1021.293,-53.472,-96.579,166.328,50.511,159.146
C06527=1021.300,-53.193,-96.591,166.331,50.506,159.145
C06528=1021.306,-52.914,-96.604,166.335,50.502,159.145
C06529=1021.313,-52.635,-96.616,166.338,50.497,159.145
C06530=1021.319,-52.385,-96.628,166.341,50.493,159.144
C06531=1021.325,-52.135,-96.638,166.343,50.488,159.144
C06532=1021.331,-51.886,-96.649,166.347,50.483,159.144
C06533=1021.337,-51.636,-96.661,166.350,50.479,159.143
C06534=1021.342,-51.387,-96.673,166.353,50.475,159.143
C06535=1021.348,-51.137,-96.684,166.356,50.470,159.143
C06536=1021.354,-50.887,-96.695,166.359,50.466,159.143
C06537=1021.359,-50.637,-96.706,166.362,50.461,159.142
C06538=1021.366,-50.388,-96.718,166.365,50.457,159.142
C06539=1021.371,-50.138,-96.730,166.367,50.453,159.142
C06540=1021.377,-49.888,-96.741,166.371,50.449,159.142
C06541=1021.383,-49.638,-96.753,166.374,50.445,159.141
C06542=1021.388,-49.389,-96.764,166.376,50.441,159.141
C06543=1021.394,-49.140,-96.776,166.379,50.437,159.141
C06544=1021.400,-48.890,-96.788,166.383,50.432,159.141
C06545=1021.405,-48.640,-96.800,166.385,50.428,159.140
C06546=1021.412,-48.390,-96.811,166.388,50.424,159.140
C06547=1021.417,-48.140,-96.822,166.392,50.420,159.140
C06548=1021.423,-47.891,-96.834,166.394,50.415,159.140
C06549=1021.428,-47.641,-96.846,166.397,50.411,159.139
C06550=1021.434,-47.392,-96.858,166.400,50.407,159.139
C06551=1021.440,-47.142,-96.869,166.403,50.403,159.139
C06552=1021.445,-46.892,-96.882,166.406,50.399,159.138
C06553=1021.451,-46.643,-96.892,166.409,50.395,159.138
C06554=1021.457,-46.393,-96.905,166.411,50.391,159.138
C06555=1021.463,-46.144,-96.916,166.415,50.386,159.138
C06556=1021.469,-45.894,-96.928,166.418,50.382,159.137
C06557=1021.474,-45.644,-96.939,166.420,50.378,159.137
C06558=1021.479,-45.429,-96.950,166.423,50.374,159.137
C06559=1021.484,-45.214,-96.960,166.426,50.370,159.137
C06560=1021.489,-44.999,-96.970,166.428,50.367,159.136
C06561=1021.494,-44.785,-96.980,166.430,50.363,159.136
C06562=1021.499,-44.570,-96.990,166.433,50.359,159.136
C06563=1021.504,-44.356,-97.000,166.435,50.355,159.135
C06564=1021.508,-44.140,-97.011,166.438,50.352,159.135
C06565=1021.514,-43.925,-97.021,166.441,50.348,159.135
C06566=1021.520,-43.676,-97.032,166.443,50.344,159.135
C06567=1021.526,-43.427,-97.045,166.446,50.340,159.135
C06568=1021.531,-43.177,-97.056,166.450,50.335,159.134
C06569=1021.537,-42.927,-97.068,166.452,50.331,159.134
C06570=1021.542,-42.677,-97.080,166.455,50.327,159.134
C06571=1021.549,-42.428,-97.092,166.459,50.323,159.134
C06572=1021.554,-42.179,-97.104,166.461,50.318,159.133
C06573=1021.561,-41.928,-97.115,166.464,50.314,159.133
C06574=1021.566,-41.679,-97.127,166.467,50.309,159.133
C06575=1021.573,-41.430,-97.139,166.470,50.305,159.132
C06576=1021.578,-41.180,-97.151,166.473,50.301,159.132
C06577=1021.584,-40.930,-97.163,166.476,50.297,159.132
C06578=1021.590,-40.681,-97.175,166.479,50.292,159.131
C06579=1021.595,-40.431,-97.187,166.481,50.288,159.131
C06580=1021.602,-40.181,-97.199,166.484,50.284,159.131
C06581=1021.607,-39.932,-97.211,166.488,50.279,159.131
C06582=1021.614,-39.682,-97.222,166.490,50.275,159.130
C06583=1021.619,-39.433,-97.234,166.493,50.271,159.130
C06584=1021.625,-39.183,-97.247,166.496,50.266,159.130
C06585=1021.630,-38.933,-97.259,166.499,50.262,159.129
C06586=1021.636,-38.683,-97.270,166.502,50.258,159.129
C06587=1021.642,-38.433,-97.283,166.504,50.254,159.129
C06588=1021.648,-38.184,-97.295,166.508,50.250,159.129
C06589=1021.653,-37.934,-97.308,166.511,50.245,159.128
C06590=1021.662,-37.586,-97.325,166.515,50.239,159.128
C06591=1021.670,-37.238,-97.341,166.519,50.234,159.128
C06592=1021.677,-36.889,-97.359,166.523,50.228,159.127
C06593=1021.685,-36.541,-97.376,166.526,50.222,159.127
C06594=1021.691,-36.291,-97.388,166.530,50.218,159.126
C06595=1021.697,-36.041,-97.401,166.533,50.214,159.126
C06596=1021.702,-35.792,-97.413,166.535,50.209,159.126
C06597=1021.709,-35.542,-97.425,166.538,50.205,159.125
C06598=1021.715,-35.292,-97.437,166.542,50.201,159.125
C06599=1021.720,-35.042,-97.449,166.544,50.197,159.125
C06600=1021.726,-34.793,-97.462,166.547,50.193,159.125
C06601=1021.732,-34.543,-97.474,166.550,50.189,159.124
C06602=1021.737,-34.293,-97.486,166.553,50.184,159.124
C06603=1021.743,-34.044,-97.499,166.556,50.180,159.124
C06604=1021.750,-33.794,-97.511,166.558,50.176,159.123
C06605=1021.755,-33.545,-97.523,166.561,50.171,159.123
C06606=1021.761,-33.295,-97.536,166.565,50.167,159.123
C06607=1021.767,-33.045,-97.548,166.567,50.163,159.123
C06608=1021.772,-32.796,-97.560,166.570,50.159,159.122
C06609=1021.778,-32.546,-97.573,166.573,50.155,159.122
C06610=1021.784,-32.296,-97.586,166.576,50.150,159.122
C06611=1021.791,-32.047,-97.597,166.579,50.146,159.121
C06612=1021.796,-31.797,-97.610,166.581,50.142,159.121
C06613=1021.802,-31.547,-97.622,166.584,50.138,159.121
C06614=1021.808,-31.298,-97.635,166.588,50.133,159.121
C06615=1021.814,-31.048,-97.648,166.590,50.129,159.120
C06616=1021.819,-30.799,-97.660,166.593,50.125,159.120
C06617=1021.825,-30.549,-97.673,166.595,50.120,159.119
C06618=1021.832,-30.300,-97.685,166.599,50.116,159.119
C06619=1021.838,-30.050,-97.697,166.602,50.112,159.119
C06620=1021.843,-29.801,-97.709,166.604,50.108,159.119
C06621=1021.849,-29.551,-97.722,166.607,50.104,159.118
C06622=1021.855,-29.301,-97.735,166.611,50.099,159.118
C06623=1021.861,-29.051,-97.747,166.613,50.095,159.118
C06624=1021.866,-28.802,-97.759,166.616,50.090,159.117
C06625=1021.872,-28.553,-97.773,166.619,50.086,159.117
C06626=1021.878,-28.303,-97.785,166.622,50.081,159.117
C06627=1021.885,-28.053,-97.797,166.625,50.077,159.116
C06628=1021.891,-27.803,-97.810,166.627,50.073,159.116
C06629=1021.896,-27.554,-97.822,166.630,50.069,159.116
C06630=1021.902,-27.304,-97.834,166.634,50.065,159.116
C06631=1021.908,-27.055,-97.848,166.636,50.061,159.115
C06632=1021.913,-26.805,-97.861,166.639,50.056,159.115
C06633=1021.919,-26.555,-97.873,166.641,50.052,159.114
C06634=1021.925,-26.305,-97.886,166.644,50.048,159.114
C06635=1021.931,-26.056,-97.899,166.648,50.043,159.114
C06636=1021.937,-25.806,-97.911,166.650,50.039,159.114
C06637=1021.943,-25.557,-97.924,166.653,50.035,159.113
C06638=1021.948,-25.307,-97.938,166.656,50.031,159.113
C06639=1021.954,-25.057,-97.950,166.658,50.027,159.113
C06640=1021.960,-24.807,-97.963,166.661,50.023,159.112
C06641=1021.966,-24.558,-97.976,166.665,50.019,159.112
C06642=1021.971,-24.309,-97.988,166.668,50.015,159.112
C06643=1021.978,-24.060,-98.002,166.670,50.010,159.111
C06644=1021.983,-23.810,-98.014,166.673,50.006,159.111
C06645=1021.989,-23.559,-98.027,166.675,50.002,159.111
C06646=1021.995,-23.310,-98.041,166.679,49.997,159.111
C06647=1022.001,-23.060,-98.053,166.682,49.993,159.110
C06648=1022.007,-22.811,-98.066,166.684,49.989,159.110
C06649=1022.012,-22.562,-98.079,166.687,49.985,159.110
C06650=1022.018,-22.312,-98.091,166.689,49.981,159.109
C06651=1022.024,-22.062,-98.105,166.692,49.976,159.109
C06652=1022.030,-21.813,-98.118,166.696,49.972,159.109
C06653=1022.036,-21.563,-98.131,166.698,49.968,159.108
C06654=1022.042,-21.284,-98.145,166.702,49.963,159.108
C06655=1022.049,-21.004,-98.160,166.704,49.959,159.108
C06656=1022.056,-20.724,-98.174,166.708,49.954,159.107
C06657=1022.062,-20.445,-98.189,166.711,49.949,159.107
C06658=1022.068,-20.195,-98.201,166.714,49.945,159.107
C06659=1022.074,-19.946,-98.215,166.717,49.941,159.106
C06660=1022.080,-19.696,-98.228,166.719,49.937,159.106
C06661=1022.086,-19.446,-98.241,166.722,49.932,159.106
C06662=1022.092,-19.197,-98.254,166.725,49.928,159.105
C06663=1022.098,-18.947,-98.267,166.728,49.924,159.105
C06664=1022.104,-18.697,-98.279,166.731,49.919,159.105
C06665=1022.109,-18.448,-98.293,166.733,49.915,159.104
C06666=1022.115,-18.198,-98.306,166.736,49.911,159.104
C06667=1022.121,-17.949,-98.319,166.739,49.906,159.104
C06668=1022.127,-17.699,-98.332,166.742,49.902,159.103
C06669=1022.134,-17.450,-98.345,166.744,49.898,159.103
C06670=1022.139,-17.199,-98.358,166.747,49.893,159.103
C06671=1022.145,-16.950,-98.371,166.751,49.889,159.102
C06672=1022.151,-16.701,-98.385,166.754,49.885,159.102
C06673=1022.157,-16.451,-98.397,166.756,49.880,159.102
C06674=1022.163,-16.202,-98.411,166.759,49.876,159.101
C06675=1022.169,-15.952,-98.423,166.761,49.872,159.101
C06676=1022.175,-15.702,-98.437,166.765,49.868,159.101
C06677=1022.181,-15.453,-98.450,166.767,49.863,159.100
C06678=1022.186,-15.203,-98.464,166.770,49.859,159.100
C06679=1022.192,-14.954,-98.477,166.773,49.855,159.100
C06680=1022.198,-14.704,-98.490,166.775,49.851,159.099
C06681=1022.204,-14.455,-98.504,166.778,49.847,159.099
C06682=1022.210,-14.205,-98.517,166.781,49.843,159.099
C06683=1022.215,-13.955,-98.530,166.783,49.839,159.098
C06684=1022.222,-13.706,-98.543,166.787,49.835,159.098
C06685=1022.227,-13.456,-98.557,166.790,49.830,159.098
C06686=1022.233,-13.207,-98.571,166.792,49.826,159.097
C06687=1022.238,-12.957,-98.584,166.795,49.822,159.097
C06688=1022.245,-12.708,-98.597,166.798,49.818,159.097
C06689=1022.250,-12.458,-98.611,166.800,49.814,159.097
C06690=1022.257,-12.208,-98.625,166.803,49.810,159.096
C06691=1022.262,-11.959,-98.638,166.806,49.805,159.096
C06692=1022.269,-11.709,-98.652,166.809,49.801,159.096
C06693=1022.274,-11.459,-98.665,166.812,49.797,159.095
C06694=1022.280,-11.210,-98.678,166.814,49.793,159.095
C06695=1022.286,-10.961,-98.691,166.817,49.788,159.095
C06696=1022.292,-10.711,-98.705,166.820,49.784,159.094
C06697=1022.298,-10.462,-98.718,166.822,49.780,159.094
C06698=1022.303,-10.212,-98.732,166.825,49.776,159.093
C06699=1022.310,-9.963,-98.746,166.829,49.771,159.093
C06700=1022.315,-9.712,-98.759,166.831,49.767,159.093
C06701=1022.322,-9.463,-98.772,166.834,49.763,159.092
C06702=1022.327,-9.213,-98.786,166.836,49.759,159.092
C06703=1022.333,-8.964,-98.800,166.839,49.755,159.092
C06704=1022.339,-8.714,-98.813,166.842,49.750,159.092
C06705=1022.345,-8.465,-98.827,166.845,49.745,159.091
C06706=1022.350,-8.215,-98.841,166.848,49.741,159.091
C06707=1022.357,-7.965,-98.854,166.851,49.737,159.091
C06708=1022.363,-7.716,-98.868,166.853,49.733,159.090
C06709=1022.369,-7.467,-98.881,166.856,49.729,159.090
C06710=1022.374,-7.217,-98.895,166.858,49.725,159.089
C06711=1022.381,-6.968,-98.908,166.861,49.721,159.089
C06712=1022.387,-6.719,-98.922,166.865,49.716,159.089
C06713=1022.393,-6.468,-98.936,166.867,49.712,159.088
C06714=1022.399,-6.219,-98.949,166.870,49.707,159.088
C06715=1022.405,-5.969,-98.963,166.873,49.703,159.088
C06716=1022.411,-5.720,-98.976,166.875,49.699,159.087
C06717=1022.416,-5.471,-98.990,166.878,49.695,159.087
C06718=1022.423,-5.189,-99.005,166.881,49.690,159.087
C06719=1022.430,-4.908,-99.021,166.884,49.685,159.086
C06720=1022.436,-4.626,-99.036,166.887,49.680,159.086
C06721=1022.443,-4.345,-99.052,166.890,49.676,159.085
C06722=1022.450,-4.095,-99.065,166.893,49.671,159.085
C06723=1022.456,-3.845,-99.079,166.895,49.667,159.085
C06724=1022.461,-3.596,-99.093,166.898,49.663,159.084
C06725=1022.467,-3.346,-99.107,166.901,49.659,159.084
C06726=1022.473,-3.097,-99.122,166.905,49.655,159.084
C06727=1022.478,-2.847,-99.136,166.907,49.650,159.083
C06728=1022.484,-2.597,-99.150,166.910,49.646,159.083
C06729=1022.490,-2.348,-99.163,166.913,49.642,159.083
C06730=1022.496,-2.099,-99.177,166.915,49.638,159.082
C06731=1022.502,-1.849,-99.192,166.918,49.634,159.082
C06732=1022.507,-1.599,-99.206,166.921,49.630,159.082
C06733=1022.513,-1.350,-99.219,166.923,49.626,159.081
C06734=1022.519,-1.101,-99.234,166.926,49.622,159.081
C06735=1022.526,-0.851,-99.248,166.929,49.618,159.081
C06736=1022.531,-0.601,-99.261,166.931,49.614,159.080
C06737=1022.537,-0.352,-99.275,166.934,49.609,159.080
C06738=1022.543,-0.102,-99.290,166.936,49.605,159.080
C06739=1022.548,0.148,-99.304,166.939,49.601,159.079
C06740=1022.554,0.397,-99.318,166.942,49.597,159.079
C06741=1022.560,0.646,-99.333,166.945,49.593,159.079
C06742=1022.566,0.896,-99.346,166.947,49.589,159.078
C06743=1022.572,1.146,-99.360,166.950,49.584,159.078
C06744=1022.578,1.395,-99.375,166.953,49.580,159.078
C06745=1022.584,1.645,-99.389,166.956,49.576,159.077
C06746=1022.589,1.894,-99.403,166.959,49.572,159.077
C06747=1022.595,2.143,-99.417,166.961,49.568,159.077
C06748=1022.601,2.394,-99.432,166.964,49.563,159.076
C06749=1022.607,2.643,-99.445,166.967,49.559,159.076
C06750=1022.613,2.892,-99.459,166.969,49.555,159.076
C06751=1022.619,3.142,-99.474,166.972,49.551,159.075
C06752=1022.625,3.391,-99.488,166.974,49.546,159.075
C06753=1022.630,3.641,-99.502,166.977,49.542,159.074
C06754=1022.637,3.891,-99.516,166.980,49.538,159.074
C06755=1022.642,4.140,-99.531,166.982,49.534,159.074
C06756=1022.649,4.389,-99.544,166.985,49.530,159.073
C06757=1022.655,4.639,-99.559,166.988,49.526,159.073
C06758=1022.660,4.888,-99.573,166.991,49.521,159.073
C06759=1022.666,5.137,-99.588,166.994,49.517,159.072
C06760=1022.672,5.388,-99.602,166.996,49.513,159.072
C06761=1022.678,5.637,-99.616,166.999,49.509,159.072
C06762=1022.684,5.887,-99.631,167.002,49.505,159.071
C06763=1022.690,6.136,-99.644,167.004,49.500,159.071
C06764=1022.696,6.385,-99.658,167.007,49.496,159.070
C06765=1022.702,6.635,-99.673,167.010,49.492,159.070
C06766=1022.708,6.884,-99.687,167.012,49.488,159.070
C06767=1022.714,7.135,-99.702,167.015,49.483,159.069
C06768=1022.720,7.384,-99.716,167.017,49.479,159.069
C06769=1022.725,7.633,-99.730,167.020,49.475,159.069
C06770=1022.732,7.883,-99.745,167.024,49.470,159.068
C06771=1022.738,8.132,-99.758,167.026,49.466,159.068
C06772=1022.744,8.382,-99.773,167.029,49.462,159.068
C06773=1022.750,8.631,-99.787,167.031,49.458,159.067
C06774=1022.756,8.881,-99.802,167.034,49.454,159.067
C06775=1022.762,9.130,-99.817,167.036,49.449,159.066
C06776=1022.768,9.380,-99.831,167.039,49.445,159.066
C06777=1022.774,9.629,-99.845,167.042,49.441,159.066
C06778=1022.780,9.879,-99.860,167.044,49.436,159.065
C06779=1022.786,10.128,-99.874,167.047,49.432,159.065
C06780=1022.792,10.378,-99.887,167.051,49.428,159.065
C06781=1022.798,10.627,-99.902,167.053,49.423,159.064
C06782=1022.805,10.911,-99.919,167.055,49.418,159.064
C06783=1022.811,11.194,-99.935,167.059,49.413,159.063
C06784=1022.818,11.477,-99.952,167.062,49.409,159.063
C06785=1022.825,11.761,-99.968,167.065,49.404,159.062
C06786=1022.831,12.010,-99.983,167.067,49.400,159.062
C06787=1022.837,12.259,-99.998,167.071,49.395,159.062
C06788=1022.844,12.509,-100.011,167.073,49.391,159.061
C06789=1022.850,12.758,-100.026,167.076,49.387,159.061
C06790=1022.856,13.007,-100.040,167.079,49.382,159.060
C06791=1022.862,13.258,-100.055,167.081,49.378,159.060
C06792=1022.868,13.506,-100.069,167.084,49.373,159.060
C06793=1022.874,13.756,-100.084,167.086,49.370,159.059
C06794=1022.880,14.005,-100.099,167.089,49.366,159.059
C06795=1022.885,14.256,-100.113,167.092,49.362,159.059
C06796=1022.891,14.505,-100.128,167.094,49.357,159.058
C06797=1022.897,14.754,-100.143,167.097,49.353,159.058
C06798=1022.904,15.004,-100.158,167.100,49.349,159.057
C06799=1022.909,15.253,-100.173,167.102,49.344,159.057
C06800=1022.916,15.503,-100.187,167.105,49.340,159.057
C06801=1022.921,15.752,-100.202,167.108,49.336,159.056
C06802=1022.927,16.002,-100.217,167.110,49.332,159.056
C06803=1022.933,16.251,-100.231,167.113,49.328,159.055
C06804=1022.939,16.501,-100.246,167.115,49.324,159.055
C06805=1022.945,16.750,-100.261,167.118,49.320,159.055
C06806=1022.951,16.999,-100.276,167.120,49.315,159.054
C06807=1022.957,17.250,-100.291,167.124,49.311,159.054
C06808=1022.962,17.499,-100.305,167.127,49.307,159.054
C06809=1022.969,17.749,-100.320,167.129,49.302,159.053
C06810=1022.975,17.997,-100.335,167.132,49.298,159.053
C06811=1022.981,18.247,-100.350,167.135,49.294,159.053
C06812=1022.987,18.497,-100.365,167.137,49.289,159.052
C06813=1022.992,18.746,-100.380,167.140,49.285,159.052
C06814=1022.999,18.996,-100.395,167.143,49.281,159.051
C06815=1023.005,19.245,-100.409,167.145,49.277,159.051
C06816=1023.011,19.494,-100.424,167.148,49.273,159.051
C06817=1023.017,19.744,-100.440,167.150,49.269,159.050
C06818=1023.022,19.993,-100.455,167.153,49.264,159.050
C06819=1023.029,20.243,-100.469,167.156,49.260,159.049
C06820=1023.034,20.492,-100.485,167.158,49.256,159.049
C06821=1023.040,20.742,-100.500,167.161,49.251,159.049
C06822=1023.047,20.992,-100.515,167.163,49.247,159.048
C06823=1023.052,21.241,-100.530,167.166,49.244,159.048
C06824=1023.058,21.490,-100.545,167.169,49.240,159.048
C06825=1023.064,21.740,-100.560,167.171,49.235,159.047
C06826=1023.069,21.989,-100.575,167.174,49.231,159.047
C06827=1023.076,22.239,-100.590,167.177,49.227,159.046
C06828=1023.082,22.489,-100.605,167.179,49.222,159.046
C06829=1023.087,22.738,-100.620,167.182,49.218,159.046
C06830=1023.094,22.988,-100.635,167.185,49.214,159.045
C06831=1023.100,23.237,-100.650,167.187,49.210,159.045
C06832=1023.105,23.487,-100.665,167.190,49.206,159.044
C06833=1023.112,23.736,-100.681,167.192,49.201,159.044
C06834=1023.118,23.985,-100.696,167.195,49.197,159.044
C06835=1023.123,24.234,-100.711,167.198,49.193,159.043
C06836=1023.130,24.484,-100.726,167.200,49.188,159.043
C06837=1023.136,24.734,-100.741,167.203,49.184,159.042
C06838=1023.141,24.983,-100.756,167.206,49.180,159.042
C06839=1023.147,25.233,-100.771,167.208,49.176,159.042
C06840=1023.154,25.482,-100.786,167.211,49.172,159.041
C06841=1023.159,25.731,-100.802,167.213,49.167,159.041
C06842=1023.165,25.981,-100.816,167.216,49.163,159.040
C06843=1023.171,26.231,-100.832,167.219,49.159,159.040
C06844=1023.177,26.480,-100.847,167.221,49.155,159.040
C06845=1023.183,26.729,-100.862,167.224,49.151,159.039
C06846=1023.189,27.014,-100.879,167.227,49.146,159.039
C06847=1023.197,27.299,-100.897,167.229,49.141,159.038
C06848=1023.204,27.584,-100.914,167.233,49.136,159.038
C06849=1023.211,27.868,-100.932,167.236,49.131,159.038
C06850=1023.216,28.118,-100.947,167.239,49.127,159.037
C06851=1023.223,28.367,-100.963,167.241,49.122,159.037
C06852=1023.228,28.617,-100.978,167.243,49.119,159.036
C06853=1023.234,28.867,-100.994,167.246,49.115,159.036
C06854=1023.240,29.115,-101.009,167.249,49.111,159.036
C06855=1023.246,29.365,-101.025,167.251,49.106,159.035
C06856=1023.252,29.614,-101.039,167.254,49.102,159.035
C06857=1023.258,29.864,-101.056,167.257,49.098,159.034
C06858=1023.263,30.113,-101.071,167.259,49.094,159.034
C06859=1023.270,30.362,-101.087,167.262,49.090,159.034
C06860=1023.275,30.612,-101.102,167.264,49.086,159.033
C06861=1023.282,30.862,-101.117,167.267,49.081,159.033
C06862=1023.288,31.111,-101.133,167.270,49.077,159.032
C06863=1023.293,31.360,-101.148,167.272,49.073,159.032
C06864=1023.299,31.609,-101.164,167.275,49.069,159.032
C06865=1023.305,31.859,-101.180,167.277,49.065,159.031
C06866=1023.311,32.109,-101.195,167.280,49.061,159.031
C06867=1023.317,32.358,-101.211,167.283,49.056,159.030
C06868=1023.323,32.607,-101.225,167.285,49.052,159.030
C06869=1023.329,32.857,-101.242,167.288,49.047,159.030
C06870=1023.335,33.107,-101.257,167.291,49.043,159.029
C06871=1023.341,33.356,-101.273,167.293,49.039,159.029
C06872=1023.347,33.606,-101.288,167.296,49.035,159.028
C06873=1023.353,33.855,-101.303,167.298,49.031,159.028
C06874=1023.359,34.104,-101.319,167.301,49.027,159.028
C06875=1023.364,34.354,-101.335,167.304,49.022,159.027
C06876=1023.371,34.603,-101.350,167.306,49.018,159.027
C06877=1023.377,34.853,-101.366,167.309,49.014,159.026
C06878=1023.383,35.102,-101.382,167.311,49.010,159.026
C06879=1023.389,35.352,-101.397,167.314,49.005,159.026
C06880=1023.394,35.601,-101.413,167.317,49.001,159.025
C06881=1023.401,35.850,-101.428,167.319,48.997,159.025
C06882=1023.407,36.100,-101.444,167.322,48.993,159.024
C06883=1023.413,36.349,-101.459,167.325,48.989,159.024
C06884=1023.419,36.599,-101.476,167.327,48.984,159.024
C06885=1023.425,36.848,-101.492,167.330,48.980,159.023
C06886=1023.431,37.098,-101.507,167.332,48.976,159.023
C06887=1023.437,37.347,-101.523,167.335,48.971,159.022
C06888=1023.442,37.596,-101.538,167.338,48.968,159.022
C06889=1023.448,37.846,-101.554,167.340,48.964,159.022
C06890=1023.454,38.095,-101.571,167.343,48.959,159.021
C06891=1023.460,38.345,-101.586,167.346,48.955,159.021
C06892=1023.466,38.594,-101.602,167.348,48.951,159.020
C06893=1023.473,38.843,-101.618,167.351,48.946,159.020
C06894=1023.478,39.093,-101.634,167.353,48.942,159.020
C06895=1023.484,39.343,-101.650,167.356,48.939,159.019
C06896=1023.490,39.592,-101.666,167.358,48.934,159.019
C06897=1023.496,39.841,-101.682,167.360,48.930,159.018
C06898=1023.501,40.091,-101.698,167.363,48.926,159.018
C06899=1023.507,40.340,-101.714,167.366,48.922,159.018
C06900=1023.514,40.589,-101.730,167.368,48.918,159.017
C06901=1023.519,40.839,-101.745,167.371,48.914,159.017
C06902=1023.525,41.088,-101.761,167.373,48.909,159.016
C06903=1023.531,41.338,-101.778,167.376,48.905,159.016
C06904=1023.537,41.587,-101.794,167.379,48.901,159.015
C06905=1023.543,41.837,-101.809,167.381,48.897,159.015
C06906=1023.549,42.086,-101.826,167.384,48.893,159.015
C06907=1023.556,42.335,-101.841,167.387,48.888,159.014
C06908=1023.562,42.585,-101.858,167.389,48.884,159.014
C06909=1023.568,42.834,-101.874,167.392,48.880,159.014
C06910=1023.574,43.119,-101.892,167.395,48.876,159.013
C06911=1023.580,43.403,-101.910,167.398,48.871,159.013
C06912=1023.587,43.688,-101.929,167.400,48.866,159.012
C06913=1023.594,43.973,-101.947,167.404,48.861,159.012
C06914=1023.599,44.222,-101.964,167.406,48.858,159.011
C06915=1023.605,44.472,-101.980,167.408,48.854,159.011
C06916=1023.611,44.721,-101.997,167.411,48.850,159.011
C06917=1023.617,44.970,-102.013,167.414,48.845,159.010
C06918=1023.623,45.220,-102.029,167.416,48.841,159.010
C06919=1023.629,45.469,-102.045,167.419,48.837,159.009
C06920=1023.634,45.718,-102.062,167.421,48.833,159.009
C06921=1023.640,45.968,-102.078,167.424,48.829,159.009
C06922=1023.646,46.218,-102.095,167.427,48.825,159.008
C06923=1023.652,46.467,-102.111,167.429,48.821,159.008
C06924=1023.658,46.716,-102.127,167.431,48.816,159.007
C06925=1023.663,46.966,-102.144,167.434,48.813,159.007
C06926=1023.669,47.215,-102.160,167.437,48.809,159.007
C06927=1023.675,47.464,-102.176,167.439,48.804,159.006
C06928=1023.681,47.714,-102.193,167.442,48.800,159.006
C06929=1023.687,47.963,-102.209,167.445,48.796,159.005
C06930=1023.692,48.213,-102.225,167.447,48.792,159.005
C06931=1023.698,48.462,-102.242,167.450,48.788,159.005
C06932=1023.704,48.711,-102.258,167.453,48.784,159.004
C06933=1023.710,48.961,-102.274,167.455,48.779,159.004
C06934=1023.716,49.210,-102.290,167.457,48.775,159.003
C06935=1023.722,49.460,-102.307,167.460,48.771,159.003
C06936=1023.727,49.709,-102.324,167.462,48.767,159.002
C06937=1023.733,49.958,-102.340,167.465,48.763,159.002
C06938=1023.739,50.208,-102.356,167.467,48.759,159.002
C06939=1023.746,50.456,-102.373,167.470,48.754,159.001
C06940=1023.752,50.706,-102.390,167.473,48.751,159.001
C06941=1023.758,50.956,-102.406,167.475,48.747,159.001
C06942=1023.763,51.205,-102.423,167.478,48.742,159.000
C06943=1023.769,51.455,-102.439,167.481,48.738,159.000
C06944=1023.775,51.704,-102.455,167.483,48.733,158.999
C06945=1023.781,51.954,-102.472,167.486,48.730,158.999
C06946=1023.787,52.203,-102.488,167.489,48.726,158.999
C06947=1023.793,52.452,-102.504,167.491,48.721,158.998
C06948=1023.799,52.701,-102.522,167.494,48.717,158.998
C06949=1023.805,52.951,-102.538,167.495,48.713,158.997
C06950=1023.811,53.200,-102.554,167.498,48.709,158.997
C06951=1023.817,53.450,-102.571,167.501,48.705,158.996
C06952=1023.823,53.699,-102.587,167.503,48.700,158.996
C06953=1023.829,53.949,-102.603,167.506,48.696,158.995
C06954=1023.834,54.198,-102.621,167.508,48.692,158.995
C06955=1023.840,54.447,-102.637,167.511,48.688,158.995
C06956=1023.846,54.696,-102.653,167.514,48.683,158.994
C06957=1023.852,54.946,-102.670,167.516,48.679,158.994
C06958=1023.859,55.196,-102.686,167.519,48.675,158.993
C06959=1023.865,55.445,-102.703,167.522,48.671,158.993
C06960=1023.870,55.694,-102.720,167.524,48.667,158.993
C06961=1023.876,55.944,-102.736,167.527,48.662,158.992
C06962=1023.882,56.193,-102.753,167.530,48.658,158.992
C06963=1023.889,56.442,-102.770,167.532,48.654,158.991
C06964=1023.895,56.692,-102.786,167.535,48.650,158.991
C06965=1023.901,56.941,-102.802,167.537,48.645,158.990
C06966=1023.906,57.191,-102.819,167.540,48.641,158.990
C06967=1023.912,57.439,-102.836,167.542,48.637,158.989
C06968=1023.918,57.689,-102.852,167.545,48.633,158.989
C06969=1023.924,57.938,-102.869,167.548,48.628,158.989
C06970=1023.931,58.188,-102.885,167.550,48.624,158.988
C06971=1023.936,58.437,-102.903,167.553,48.620,158.988
C06972=1023.942,58.687,-102.919,167.556,48.616,158.987
C06973=1023.948,58.936,-102.935,167.558,48.611,158.987
C06974=1023.956,59.220,-102.955,167.561,48.607,158.986
C06975=1023.962,59.504,-102.974,167.564,48.602,158.986
C06976=1023.969,59.789,-102.993,167.566,48.597,158.985
C06977=1023.976,60.074,-103.011,167.570,48.592,158.985
C06978=1023.983,60.323,-103.029,167.572,48.588,158.984
C06979=1023.989,60.572,-103.045,167.575,48.584,158.984
C06980=1023.994,60.822,-103.062,167.578,48.579,158.984
C06981=1024.000,61.071,-103.079,167.580,48.575,158.983
C06982=1024.007,61.321,-103.095,167.583,48.571,158.983
C06983=1024.013,61.570,-103.112,167.585,48.566,158.982
C06984=1024.019,61.819,-103.129,167.588,48.562,158.982
C06985=1024.025,62.068,-103.145,167.591,48.558,158.981
C06986=1024.031,62.318,-103.163,167.593,48.554,158.981
C06987=1024.037,62.567,-103.179,167.596,48.549,158.980
C06988=1024.043,62.817,-103.195,167.598,48.545,158.980
C06989=1024.050,63.066,-103.213,167.601,48.541,158.980
C06990=1024.055,63.316,-103.230,167.603,48.536,158.979
C06991=1024.061,63.564,-103.247,167.606,48.532,158.979
C06992=1024.066,63.814,-103.263,167.608,48.529,158.978
C06993=1024.073,64.063,-103.281,167.610,48.524,158.978
C06994=1024.079,64.313,-103.298,167.613,48.520,158.977
C06995=1024.085,64.562,-103.315,167.616,48.516,158.977
C06996=1024.091,64.812,-103.332,167.618,48.512,158.977
C06997=1024.097,65.061,-103.349,167.621,48.507,158.976
C06998=1024.102,65.310,-103.366,167.624,48.503,158.976
C06999=1024.108,65.559,-103.383,167.626,48.499,158.975
C07000=1024.114,65.809,-103.400,167.629,48.495,158.975
C07001=1024.120,66.058,-103.417,167.632,48.491,158.974
C07002=1024.126,66.307,-103.434,167.634,48.486,158.974
C07003=1024.133,66.557,-103.452,167.637,48.482,158.974
C07004=1024.138,66.807,-103.468,167.639,48.478,158.973
C07005=1024.144,67.055,-103.485,167.642,48.474,158.973
C07006=1024.150,67.305,-103.503,167.644,48.470,158.972
C07007=1024.156,67.554,-103.520,167.646,48.466,158.972
C07008=1024.162,67.803,-103.537,167.649,48.462,158.971
C07009=1024.169,68.053,-103.555,167.652,48.457,158.971
C07010=1024.174,68.303,-103.571,167.654,48.453,158.971
C07011=1024.179,68.552,-103.589,167.657,48.449,158.970
C07012=1024.186,68.801,-103.606,167.660,48.445,158.970
C07013=1024.191,69.051,-103.623,167.663,48.441,158.969
C07014=1024.197,69.300,-103.641,167.665,48.437,158.969
C07015=1024.204,69.549,-103.658,167.668,48.433,158.968
C07016=1024.209,69.798,-103.676,167.670,48.428,158.968
C07017=1024.215,70.048,-103.692,167.673,48.424,158.968
C07018=1024.221,70.297,-103.710,167.676,48.420,158.967
C07019=1024.227,70.546,-103.727,167.677,48.416,158.967
C07020=1024.232,70.795,-103.745,167.680,48.412,158.966
C07021=1024.239,71.045,-103.762,167.682,48.408,158.966
C07022=1024.245,71.294,-103.779,167.685,48.404,158.965
C07023=1024.250,71.543,-103.797,167.688,48.400,158.965
C07024=1024.256,71.793,-103.815,167.691,48.395,158.965
C07025=1024.262,72.042,-103.832,167.693,48.391,158.964
C07026=1024.269,72.292,-103.850,167.696,48.387,158.964
C07027=1024.274,72.541,-103.866,167.699,48.383,158.963
C07028=1024.279,72.790,-103.884,167.701,48.378,158.963
C07029=1024.286,73.040,-103.901,167.704,48.374,158.962
C07030=1024.292,73.289,-103.919,167.707,48.371,158.962
C07031=1024.298,73.539,-103.937,167.708,48.366,158.961
C07032=1024.304,73.787,-103.954,167.711,48.362,158.961
C07033=1024.310,74.036,-103.971,167.713,48.358,158.961
C07034=1024.316,74.286,-103.989,167.716,48.354,158.960
C07035=1024.321,74.536,-104.006,167.719,48.349,158.960
C07036=1024.328,74.785,-104.023,167.721,48.346,158.959
C07037=1024.333,75.034,-104.041,167.724,48.342,158.959
C07038=1024.340,75.319,-104.061,167.727,48.336,158.958
C07039=1024.347,75.602,-104.081,167.730,48.332,158.958
C07040=1024.353,75.887,-104.101,167.733,48.327,158.957
C07041=1024.360,76.172,-104.121,167.736,48.322,158.957
C07042=1024.366,76.420,-104.138,167.739,48.318,158.957
C07043=1024.372,76.670,-104.156,167.741,48.314,158.956
C07044=1024.378,76.919,-104.174,167.744,48.310,158.956
C07045=1024.384,77.169,-104.192,167.747,48.306,158.955
C07046=1024.390,77.418,-104.209,167.749,48.301,158.955
C07047=1024.396,77.668,-104.227,167.752,48.298,158.954
C07048=1024.401,77.917,-104.245,167.753,48.293,158.954
C07049=1024.407,78.166,-104.263,167.756,48.289,158.954
C07050=1024.413,78.415,-104.281,167.759,48.286,158.953
C07051=1024.419,78.664,-104.299,167.761,48.281,158.953
C07052=1024.425,78.914,-104.316,167.764,48.277,158.952
C07053=1024.430,79.163,-104.334,167.767,48.273,158.952
C07054=1024.437,79.412,-104.352,167.770,48.269,158.951
C07055=1024.442,79.661,-104.370,167.772,48.265,158.951
C07056=1024.448,79.911,-104.387,167.775,48.261,158.951
C07057=1024.454,80.160,-104.405,167.777,48.257,158.950
C07058=1024.460,80.409,-104.424,167.779,48.253,158.950
C07059=1024.466,80.658,-104.441,167.782,48.248,158.949
C07060=1024.472,80.908,-104.459,167.785,48.244,158.949
C07061=1024.477,81.157,-104.477,167.787,48.241,158.949
C07062=1024.483,81.407,-104.495,167.790,48.236,158.948
C07063=1024.489,81.656,-104.512,167.793,48.232,158.948
C07064=1024.495,81.905,-104.531,167.796,48.228,158.947
C07065=1024.501,82.154,-104.548,167.798,48.224,158.947
C07066=1024.507,82.404,-104.566,167.801,48.220,158.946
C07067=1024.512,82.653,-104.584,167.802,48.216,158.946
C07068=1024.519,82.903,-104.602,167.805,48.212,158.945
C07069=1024.524,83.151,-104.620,167.808,48.208,158.945
C07070=1024.531,83.401,-104.638,167.810,48.203,158.945
C07071=1024.536,83.650,-104.656,167.813,48.200,158.944
C07072=1024.542,83.900,-104.674,167.816,48.195,158.944
C07073=1024.548,84.148,-104.692,167.818,48.191,158.943
C07074=1024.554,84.398,-104.710,167.821,48.187,158.943
C07075=1024.560,84.647,-104.728,167.824,48.183,158.942
C07076=1024.566,84.896,-104.745,167.827,48.179,158.942
C07077=1024.572,85.146,-104.764,167.829,48.174,158.942
C07078=1024.578,85.395,-104.782,167.832,48.171,158.941
C07079=1024.584,85.644,-104.799,167.834,48.166,158.941
C07080=1024.589,85.893,-104.817,167.837,48.162,158.940
C07081=1024.595,86.143,-104.836,167.840,48.158,158.940
C07082=1024.601,86.393,-104.854,167.841,48.154,158.939
C07083=1024.607,86.642,-104.872,167.844,48.149,158.939
C07084=1024.613,86.891,-104.890,167.847,48.146,158.938
C07085=1024.619,87.140,-104.908,167.849,48.141,158.938
C07086=1024.625,87.390,-104.926,167.852,48.137,158.938
C07087=1024.631,87.639,-104.945,167.855,48.133,158.937
C07088=1024.637,87.888,-104.962,167.857,48.129,158.937
C07089=1024.643,88.137,-104.980,167.860,48.125,158.936
C07090=1024.649,88.386,-104.998,167.863,48.120,158.936
C07091=1024.655,88.636,-105.016,167.865,48.117,158.935
C07092=1024.661,88.885,-105.034,167.868,48.112,158.935
C07093=1024.667,89.134,-105.052,167.871,48.108,158.935
C07094=1024.673,89.384,-105.070,167.873,48.104,158.934
C07095=1024.679,89.633,-105.089,167.876,48.100,158.934
C07096=1024.684,89.882,-105.107,167.879,48.095,158.933
C07097=1024.690,90.131,-105.126,167.881,48.091,158.933
C07098=1024.696,90.381,-105.144,167.884,48.088,158.932
C07099=1024.702,90.630,-105.163,167.887,48.083,158.932
C07100=1024.708,90.879,-105.181,167.888,48.080,158.931
C07101=1024.713,91.128,-105.200,167.891,48.076,158.931
C07102=1024.720,91.413,-105.220,167.895,48.071,158.931
C07103=1024.727,91.697,-105.241,167.897,48.066,158.930
C07104=1024.733,91.981,-105.262,167.901,48.062,158.930
C07105=1024.740,92.265,-105.283,167.903,48.057,158.929
C07106=1024.746,92.515,-105.301,167.906,48.053,158.929
C07107=1024.752,92.764,-105.320,167.909,48.049,158.928
C07108=1024.757,93.013,-105.338,167.911,48.045,158.928
C07109=1024.763,93.262,-105.357,167.914,48.040,158.927
C07110=1024.769,93.512,-105.376,167.917,48.036,158.927
C07111=1024.775,93.761,-105.394,167.920,48.033,158.927
C07112=1024.781,94.010,-105.412,167.922,48.028,158.926
C07113=1024.786,94.260,-105.431,167.925,48.024,158.926
C07114=1024.792,94.508,-105.449,167.926,48.020,158.925
C07115=1024.799,94.757,-105.468,167.929,48.016,158.925
C07116=1024.804,95.007,-105.486,167.932,48.012,158.924
C07117=1024.810,95.256,-105.505,167.934,48.008,158.924
C07118=1024.816,95.505,-105.523,167.937,48.004,158.924
C07119=1024.822,95.755,-105.542,167.940,48.000,158.923
C07120=1024.828,96.003,-105.560,167.943,47.996,158.923
C07121=1024.834,96.253,-105.579,167.945,47.992,158.922
C07122=1024.839,96.503,-105.597,167.948,47.987,158.922
C07123=1024.846,96.752,-105.616,167.951,47.983,158.921
C07124=1024.851,97.000,-105.635,167.953,47.979,158.921
C07125=1024.857,97.250,-105.653,167.956,47.975,158.921
C07126=1024.863,97.499,-105.671,167.959,47.971,158.920
C07127=1024.869,97.749,-105.691,167.961,47.967,158.920
C07128=1024.875,97.998,-105.708,167.964,47.963,158.919
C07129=1024.881,98.247,-105.727,167.967,47.958,158.919
C07130=1024.887,98.496,-105.746,167.970,47.955,158.918
C07131=1024.893,98.745,-105.765,167.972,47.950,158.918
C07132=1024.899,98.995,-105.782,167.975,47.946,158.918
C07133=1024.904,99.244,-105.801,167.977,47.942,158.917
C07134=1024.911,99.493,-105.820,167.980,47.938,158.917
C07135=1024.917,99.743,-105.839,167.983,47.933,158.916
C07136=1024.923,99.992,-105.858,167.986,47.930,158.916
C07137=1024.928,100.241,-105.876,167.987,47.926,158.915
C07138=1024.933,100.490,-105.895,167.990,47.922,158.915
C07139=1024.940,100.740,-105.914,167.993,47.918,158.914
C07140=1024.946,100.989,-105.933,167.996,47.914,158.914
C07141=1024.951,101.238,-105.952,167.998,47.910,158.914
C07142=1024.957,101.487,-105.971,168.001,47.906,158.913
C07143=1024.963,101.736,-105.990,168.004,47.902,158.913
C07144=1024.968,101.986,-106.009,168.007,47.898,158.912
C07145=1024.975,102.235,-106.028,168.009,47.893,158.912
C07146=1024.980,102.484,-106.047,168.012,47.890,158.912
C07147=1024.986,102.733,-106.066,168.015,47.886,158.911
C07148=1024.992,102.983,-106.084,168.017,47.881,158.911
C07149=1024.997,103.232,-106.103,168.020,47.877,158.910
C07150=1025.003,103.482,-106.123,168.023,47.874,158.910
C07151=1025.009,103.730,-106.141,168.024,47.869,158.909
C07152=1025.015,103.979,-106.160,168.027,47.866,158.909
C07153=1025.021,104.229,-106.179,168.030,47.862,158.909
C07154=1025.027,104.478,-106.198,168.033,47.857,158.908
C07155=1025.032,104.727,-106.217,168.035,47.853,158.908
C07156=1025.038,104.976,-106.235,168.038,47.849,158.907
C07157=1025.044,105.225,-106.255,168.041,47.845,158.907
C07158=1025.050,105.475,-106.274,168.044,47.841,158.906
C07159=1025.056,105.724,-106.293,168.046,47.837,158.906
C07160=1025.062,105.973,-106.312,168.049,47.833,158.906
C07161=1025.067,106.223,-106.331,168.052,47.829,158.905
C07162=1025.074,106.471,-106.350,168.054,47.825,158.905
C07163=1025.079,106.720,-106.369,168.057,47.821,158.904
C07164=1025.085,106.969,-106.389,168.060,47.816,158.904
C07165=1025.091,107.218,-106.407,168.062,47.813,158.903
C07166=1025.098,107.503,-106.429,168.065,47.808,158.903
C07167=1025.104,107.788,-106.451,168.068,47.803,158.902
C07168=1025.111,108.072,-106.472,168.072,47.799,158.902
C07169=1025.118,108.355,-106.494,168.075,47.794,158.901
C07170=1025.124,108.605,-106.513,168.077,47.790,158.901
C07171=1025.129,108.854,-106.533,168.080,47.786,158.901
C07172=1025.136,109.103,-106.551,168.083,47.782,158.900
C07173=1025.141,109.353,-106.571,168.085,47.777,158.900
C07174=1025.147,109.602,-106.590,168.088,47.774,158.899
C07175=1025.154,109.851,-106.608,168.091,47.770,158.899
C07176=1025.160,110.100,-106.628,168.093,47.765,158.898
C07177=1025.165,110.350,-106.648,168.096,47.762,158.898
C07178=1025.171,110.599,-106.667,168.099,47.758,158.898
C07179=1025.177,110.848,-106.686,168.102,47.753,158.897
C07180=1025.183,111.097,-106.706,168.104,47.749,158.897
C07181=1025.189,111.346,-106.725,168.107,47.746,158.896
C07182=1025.194,111.595,-106.744,168.110,47.741,158.896
C07183=1025.200,111.845,-106.763,168.113,47.737,158.895
C07184=1025.206,112.093,-106.783,168.115,47.734,158.895
C07185=1025.212,112.343,-106.802,168.118,47.729,158.895
C07186=1025.217,112.592,-106.821,168.121,47.725,158.894
C07187=1025.223,112.842,-106.841,168.124,47.721,158.894
C07188=1025.229,113.090,-106.860,168.126,47.717,158.893
C07189=1025.235,113.340,-106.880,168.129,47.713,158.893
C07190=1025.241,113.589,-106.900,168.132,47.709,158.893
C07191=1025.246,113.838,-106.919,168.134,47.706,158.892
C07192=1025.252,114.088,-106.938,168.137,47.702,158.892
C07193=1025.257,114.337,-106.959,168.139,47.698,158.891
C07194=1025.263,114.586,-106.978,168.142,47.694,158.891
C07195=1025.269,114.835,-106.998,168.145,47.690,158.890
C07196=1025.275,115.084,-107.017,168.148,47.686,158.890
C07197=1025.281,115.333,-107.037,168.150,47.682,158.890
